LIN {X 0,Y 572.963,Z 548.941,A -85,B 0,C 180,E1 -2254.928,E2 -2254.928} C_VEL
LIN {X 0,Y 573.068,Z 542.866,A -85,B 0,C 180,E1 -2256.162,E2 -2256.162} C_VEL
LIN {X 0,Y 573.121,Z 536.225,A -85,B 0,C 180,E1 -2257.223,E2 -2257.223} C_VEL
LIN {X 0,Y 573.193,Z 527.976,A -85,B 0,C 180,E1 -2258.285,E2 -2258.285} C_VEL
LIN {X 0,Y 573.321,Z 517.583,A -85,B 0,C 180,E1 -2259.349,E2 -2259.349} C_VEL
LIN {X 0,Y 573.439,Z 507.903,A -85,B 0,C 180,E1 -2260.149,E2 -2260.149} C_VEL
LIN {X 0,Y 573.55,Z 497.379,A -85,B 0,C 180,E1 -2260.856,E2 -2260.856} C_VEL
LIN {X 0,Y 573.652,Z 485.088,A -85,B 0,C 180,E1 -2261.502,E2 -2261.502} C_VEL
LIN {X 0,Y 573.708,Z 473.128,A -85,B 0,C 180,E1 -2261.977,E2 -2261.977} C_VEL
LIN {X 0,Y 573.816,Z 460.458,A -85,B 0,C 180,E1 -2262.333,E2 -2262.333} C_VEL
LIN {X 0,Y 573.909,Z 447.193,A -85,B 0,C 180,E1 -2262.556,E2 -2262.556} C_VEL
LIN {X 0,Y 573.954,Z 350.61,A -85,B 0,C 180,E1 -2263.77,E2 -2263.77} C_VEL
LIN {X 0,Y 573.392,Z 346.603,A -85,B 0,C 180,E1 -2263.852,E2 -2263.852} C_VEL
LIN {X 0,Y 573.571,Z 326.113,A -85,B 0,C 180,E1 -2266.728,E2 -2266.728} C_VEL
LIN {X 0,Y 573.806,Z 305.604,A -85,B 0,C 180,E1 -2269.647,E2 -2269.647} C_VEL
LIN {X 0,Y 574.031,Z 285.779,A -85,B 0,C 180,E1 -2272.496,E2 -2272.496} C_VEL
LIN {X 0,Y 573.584,Z 280.847,A -85,B 0,C 180,E1 -2273.225,E2 -2273.225} C_VEL
LIN {X 0,Y 573.243,Z 279.081,A -85,B 0,C 180,E1 -2273.497,E2 -2273.497} C_VEL
LIN {X 0,Y 573.263,Z 279.079,A -85,B 0,C 180,E1 -2276.19,E2 -2276.19} C_VEL
LIN {X 0,Y 573.238,Z 279.077,A -85,B 0,C 180,E1 -2278.565,E2 -2278.565} C_VEL
LIN {X 0,Y 573.228,Z 279.075,A -85,B 0,C 180,E1 -2280.993,E2 -2280.993} C_VEL
LIN {X 0,Y 573.265,Z 279.072,A -85,B 0,C 180,E1 -2283.524,E2 -2283.524} C_VEL
LIN {X 0,Y 573.216,Z 279.084,A -85,B 0,C 180,E1 -2286.051,E2 -2286.051} C_VEL
LIN {X 0,Y 573.242,Z 279.076,A -85,B 0,C 180,E1 -2288.701,E2 -2288.701} C_VEL
LIN {X 0,Y 573.243,Z 279.073,A -85,B 0,C 180,E1 -2291.594,E2 -2291.594} C_VEL
LIN {X 0,Y 573.222,Z 279.085,A -85,B 0,C 180,E1 -2294.334,E2 -2294.334} C_VEL
LIN {X 0,Y 573.237,Z 279.074,A -85,B 0,C 180,E1 -2297.358,E2 -2297.358} C_VEL
LIN {X 0,Y 573.242,Z 279.081,A -85,B 0,C 180,E1 -2300.392,E2 -2300.392} C_VEL
LIN {X 0,Y 573.25,Z 279.075,A -85,B 0,C 180,E1 -2303.077,E2 -2303.077} C_VEL
LIN {X 0,Y 573.261,Z 279.07,A -85,B 0,C 180,E1 -2305.671,E2 -2305.671} C_VEL
LIN {X 0,Y 573.241,Z 279.075,A -85,B 0,C 180,E1 -2308.184,E2 -2308.184} C_VEL
LIN {X 0,Y 573.26,Z 279.079,A -85,B 0,C 180,E1 -2310.634,E2 -2310.634} C_VEL
LIN {X 0,Y 573.262,Z 279.072,A -85,B 0,C 180,E1 -2313.5,E2 -2313.5} C_VEL
LIN {X 0,Y 573.222,Z 279.076,A -85,B 0,C 180,E1 -2316.134,E2 -2316.134} C_VEL
LIN {X 0,Y 573.238,Z 279.081,A -85,B 0,C 180,E1 -2319.173,E2 -2319.173} C_VEL
LIN {X 0,Y 573.216,Z 279.081,A -85,B 0,C 180,E1 -2321.411,E2 -2321.411} C_VEL
LIN {X 0,Y 573.235,Z 279.076,A -85,B 0,C 180,E1 -2323.621,E2 -2323.621} C_VEL
LIN {X 0,Y 573.259,Z 279.072,A -85,B 0,C 180,E1 -2325.807,E2 -2325.807} C_VEL
LIN {X 0,Y 573.27,Z 279.072,A -85,B 0,C 180,E1 -2328.734,E2 -2328.734} C_VEL
LIN {X 0,Y 573.264,Z 279.076,A -85,B 0,C 180,E1 -2331.54,E2 -2331.54} C_VEL
LIN {X 0,Y 573.275,Z 279.069,A -85,B 0,C 180,E1 -2334.372,E2 -2334.372} C_VEL
LIN {X 0,Y 573.303,Z 279.072,A -85,B 0,C 180,E1 -2337.189,E2 -2337.189} C_VEL
LIN {X 0,Y 573.294,Z 279.069,A -85,B 0,C 180,E1 -2340,E2 -2340} C_VEL
LIN {X 0,Y 573.287,Z 279.068,A -85,B 0,C 180,E1 -2342.811,E2 -2342.811} C_VEL
LIN {X 0,Y 573.277,Z 279.08,A -85,B 0,C 180,E1 -2345.628,E2 -2345.628} C_VEL
LIN {X 0,Y 573.238,Z 279.074,A -85,B 0,C 180,E1 -2348.46,E2 -2348.46} C_VEL
LIN {X 0,Y 573.258,Z 279.074,A -85,B 0,C 180,E1 -2351.312,E2 -2351.312} C_VEL
LIN {X 0,Y 573.246,Z 279.074,A -85,B 0,C 180,E1 -2354.416,E2 -2354.416} C_VEL
LIN {X 0,Y 573.237,Z 279.074,A -85,B 0,C 180,E1 -2357.112,E2 -2357.112} C_VEL
LIN {X 0,Y 573.222,Z 279.084,A -85,B 0,C 180,E1 -2360.078,E2 -2360.078} C_VEL
LIN {X 0,Y 573.206,Z 279.082,A -85,B 0,C 180,E1 -2362.339,E2 -2362.339} C_VEL
LIN {X 0,Y 573.21,Z 279.079,A -85,B 0,C 180,E1 -2364.365,E2 -2364.365} C_VEL
LIN {X 0,Y 572.569,Z 279.16,A -85,B 0,C 180,E1 -2364.951,E2 -2364.951} C_VEL
LIN {X 0,Y 569.724,Z 279.518,A -85,B 0,C 180,E1 -2365.903,E2 -2365.903} C_VEL
LIN {X 0,Y 567.294,Z 279.816,A -85,B 0,C 180,E1 -2366.668,E2 -2366.668} C_VEL
LIN {X 0,Y 566.235,Z 279.946,A -85,B 0,C 180,E1 -2367.259,E2 -2367.259} C_VEL
LIN {X 0,Y 566.142,Z 279.958,A -85,B 0,C 180,E1 -2367.459,E2 -2367.459} C_VEL
LIN {X 0,Y 566.163,Z 279.959,A -85,B 0,C 180,E1 -2370.594,E2 -2370.594} C_VEL
LIN {X 0,Y 566.19,Z 279.952,A -85,B 0,C 180,E1 -2373.104,E2 -2373.104} C_VEL
LIN {X 0,Y 566.129,Z 279.96,A -85,B 0,C 180,E1 -2375.695,E2 -2375.695} C_VEL
LIN {X 0,Y 566.191,Z 279.959,A -85,B 0,C 180,E1 -2378.557,E2 -2378.557} C_VEL
LIN {X 0,Y 566.124,Z 279.961,A -85,B 0,C 180,E1 -2381.144,E2 -2381.144} C_VEL
LIN {X 0,Y 566.141,Z 279.96,A -85,B 0,C 180,E1 -2384.042,E2 -2384.042} C_VEL
LIN {X 0,Y 566.138,Z 279.961,A -85,B 0,C 180,E1 -2387.09,E2 -2387.09} C_VEL
LIN {X 0,Y 566.171,Z 279.958,A -85,B 0,C 180,E1 -2390.32,E2 -2390.32} C_VEL
LIN {X 0,Y 566.136,Z 279.959,A -85,B 0,C 180,E1 -2393.425,E2 -2393.425} C_VEL
LIN {X 0,Y 566.144,Z 279.959,A -85,B 0,C 180,E1 -2396.277,E2 -2396.277} C_VEL
LIN {X 0,Y 566.166,Z 279.965,A -85,B 0,C 180,E1 -2398.928,E2 -2398.928} C_VEL
LIN {X 0,Y 566.143,Z 279.957,A -85,B 0,C 180,E1 -2401.853,E2 -2401.853} C_VEL
LIN {X 0,Y 566.164,Z 279.955,A -85,B 0,C 180,E1 -2404.248,E2 -2404.248} C_VEL
LIN {X 0,Y 566.154,Z 279.962,A -85,B 0,C 180,E1 -2407.367,E2 -2407.367} C_VEL
LIN {X 0,Y 566.202,Z 279.952,A -85,B 0,C 180,E1 -2409.661,E2 -2409.661} C_VEL
LIN {X 0,Y 566.176,Z 279.955,A -85,B 0,C 180,E1 -2412.666,E2 -2412.666} C_VEL
LIN {X 0,Y 566.214,Z 279.953,A -85,B 0,C 180,E1 -2415.625,E2 -2415.625} C_VEL
LIN {X 0,Y 566.24,Z 279.946,A -85,B 0,C 180,E1 -2418.675,E2 -2418.675} C_VEL
LIN {X 0,Y 566.193,Z 279.962,A -85,B 0,C 180,E1 -2421.432,E2 -2421.432} C_VEL
LIN {X 0,Y 566.234,Z 279.946,A -85,B 0,C 180,E1 -2424.3,E2 -2424.3} C_VEL
LIN {X 0,Y 566.278,Z 279.946,A -85,B 0,C 180,E1 -2427.864,E2 -2427.864} C_VEL
LIN {X 0,Y 566.288,Z 279.944,A -85,B 0,C 180,E1 -2429.998,E2 -2429.998} C_VEL
LIN {X 0,Y 566.247,Z 279.944,A -85,B 0,C 180,E1 -2432.843,E2 -2432.843} C_VEL
LIN {X 0,Y 566.244,Z 279.954,A -85,B 0,C 180,E1 -2435.696,E2 -2435.696} C_VEL
LIN {X 0,Y 566.201,Z 279.952,A -85,B 0,C 180,E1 -2438.563,E2 -2438.563} C_VEL
LIN {X 0,Y 566.194,Z 279.956,A -85,B 0,C 180,E1 -2441.452,E2 -2441.452} C_VEL
LIN {X 0,Y 566.245,Z 280.006,A -85,B 0,C 180,E1 -2442.86,E2 -2442.86} C_VEL
LIN {X 0,Y 566.448,Z 288.153,A -85,B 0,C 180,E1 -2444.364,E2 -2444.364} C_VEL
LIN {X 0,Y 566.29,Z 303.331,A -85,B 0,C 180,E1 -2447.133,E2 -2447.133} C_VEL
LIN {X 0,Y 566.23,Z 308.399,A -85,B 0,C 180,E1 -2448.05,E2 -2448.05} C_VEL
LIN {X 0,Y 567.175,Z 314.711,A -85,B 0,C 180,E1 -2448.159,E2 -2448.159} C_VEL
LIN {X 0,Y 566.915,Z 415.457,A -85,B 0,C 180,E1 -2449.457,E2 -2449.457} C_VEL
LIN {X 0,Y 566.84,Z 428.654,A -85,B 0,C 180,E1 -2449.777,E2 -2449.777} C_VEL
LIN {X 0,Y 566.74,Z 440.771,A -85,B 0,C 180,E1 -2450.209,E2 -2450.209} C_VEL
LIN {X 0,Y 566.578,Z 452.89,A -85,B 0,C 180,E1 -2450.794,E2 -2450.794} C_VEL
LIN {X 0,Y 566.394,Z 463.739,A -85,B 0,C 180,E1 -2451.467,E2 -2451.467} C_VEL
LIN {X 0,Y 566.282,Z 474.893,A -85,B 0,C 180,E1 -2452.334,E2 -2452.334} C_VEL
LIN {X 0,Y 566.196,Z 484.666,A -85,B 0,C 180,E1 -2453.286,E2 -2453.286} C_VEL
LIN {X 0,Y 566.085,Z 493.699,A -85,B 0,C 180,E1 -2454.377,E2 -2454.377} C_VEL
LIN {X 0,Y 565.999,Z 500.298,A -85,B 0,C 180,E1 -2455.36,E2 -2455.36} C_VEL
LIN {X 0,Y 565.956,Z 506.681,A -85,B 0,C 180,E1 -2456.55,E2 -2456.55} C_VEL
LIN {X 0,Y 565.879,Z 511.585,A -85,B 0,C 180,E1 -2457.745,E2 -2457.745} C_VEL
LIN {X 0,Y 565.883,Z 515.239,A -85,B 0,C 180,E1 -2458.966,E2 -2458.966} C_VEL
LIN {X 0,Y 565.858,Z 516.997,A -85,B 0,C 180,E1 -2459.784,E2 -2459.784} C_VEL
LIN {X 0,Y 565.856,Z 518.576,A -85,B 0,C 180,E1 -2461.019,E2 -2461.019} C_VEL
LIN {X 0,Y 565.833,Z 518.934,A -85,B 0,C 180,E1 -2462.37,E2 -2462.37} C_VEL
LIN {X 0,Y 565.863,Z 517.946,A -85,B 0,C 180,E1 -2463.681,E2 -2463.681} C_VEL
LIN {X 0,Y 565.848,Z 515.692,A -85,B 0,C 180,E1 -2464.941,E2 -2464.941} C_VEL
LIN {X 0,Y 565.913,Z 512.179,A -85,B 0,C 180,E1 -2466.174,E2 -2466.174} C_VEL
LIN {X 0,Y 565.949,Z 506.981,A -85,B 0,C 180,E1 -2467.474,E2 -2467.474} C_VEL
LIN {X 0,Y 565.992,Z 500.618,A -85,B 0,C 180,E1 -2468.678,E2 -2468.678} C_VEL
LIN {X 0,Y 566.057,Z 494.058,A -85,B 0,C 180,E1 -2469.666,E2 -2469.666} C_VEL
LIN {X 0,Y 566.174,Z 484.874,A -85,B 0,C 180,E1 -2470.782,E2 -2470.782} C_VEL
LIN {X 0,Y 566.318,Z 475.145,A -85,B 0,C 180,E1 -2471.734,E2 -2471.734} C_VEL
LIN {X 0,Y 566.41,Z 464.873,A -85,B 0,C 180,E1 -2472.543,E2 -2472.543} C_VEL
LIN {X 0,Y 566.558,Z 453.576,A -85,B 0,C 180,E1 -2473.257,E2 -2473.257} C_VEL
LIN {X 0,Y 566.73,Z 441.453,A -85,B 0,C 180,E1 -2473.853,E2 -2473.853} C_VEL
LIN {X 0,Y 566.855,Z 428.486,A -85,B 0,C 180,E1 -2474.318,E2 -2474.318} C_VEL
LIN {X 0,Y 566.929,Z 414.948,A -85,B 0,C 180,E1 -2474.643,E2 -2474.643} C_VEL
LIN {X 0,Y 567.03,Z 313.172,A -85,B 0,C 180,E1 -2475.954,E2 -2475.954} C_VEL
LIN {X 0,Y 566.221,Z 308.405,A -85,B 0,C 180,E1 -2476.039,E2 -2476.039} C_VEL
LIN {X 0,Y 566.38,Z 293.821,A -85,B 0,C 180,E1 -2478.687,E2 -2478.687} C_VEL
LIN {X 0,Y 566.4,Z 281.479,A -85,B 0,C 180,E1 -2480.935,E2 -2480.935} C_VEL
LIN {X 0,Y 566.214,Z 279.954,A -85,B 0,C 180,E1 -2481.208,E2 -2481.208} C_VEL
LIN {X 0,Y 566.173,Z 279.964,A -85,B 0,C 180,E1 -2484.308,E2 -2484.308} C_VEL
LIN {X 0,Y 566.186,Z 279.954,A -85,B 0,C 180,E1 -2486.895,E2 -2486.895} C_VEL
LIN {X 0,Y 566.151,Z 279.957,A -85,B 0,C 180,E1 -2489.405,E2 -2489.405} C_VEL
LIN {X 0,Y 566.18,Z 279.956,A -85,B 0,C 180,E1 -2491.856,E2 -2491.856} C_VEL
LIN {X 0,Y 566.185,Z 279.962,A -85,B 0,C 180,E1 -2494.249,E2 -2494.249} C_VEL
LIN {X 0,Y 566.143,Z 279.965,A -85,B 0,C 180,E1 -2496.71,E2 -2496.71} C_VEL
LIN {X 0,Y 566.162,Z 279.956,A -85,B 0,C 180,E1 -2499.661,E2 -2499.661} C_VEL
LIN {X 0,Y 566.15,Z 279.965,A -85,B 0,C 180,E1 -2502.667,E2 -2502.667} C_VEL
LIN {X 0,Y 566.178,Z 279.953,A -85,B 0,C 180,E1 -2505.625,E2 -2505.625} C_VEL
LIN {X 0,Y 566.22,Z 279.958,A -85,B 0,C 180,E1 -2508.652,E2 -2508.652} C_VEL
LIN {X 0,Y 566.176,Z 279.954,A -85,B 0,C 180,E1 -2511.433,E2 -2511.433} C_VEL
LIN {X 0,Y 566.214,Z 279.952,A -85,B 0,C 180,E1 -2514.301,E2 -2514.301} C_VEL
LIN {X 0,Y 566.226,Z 279.952,A -85,B 0,C 180,E1 -2517.154,E2 -2517.154} C_VEL
LIN {X 0,Y 566.225,Z 279.946,A -85,B 0,C 180,E1 -2520,E2 -2520} C_VEL
LIN {X 0,Y 566.233,Z 279.956,A -85,B 0,C 180,E1 -2522.846,E2 -2522.846} C_VEL
LIN {X 0,Y 566.218,Z 279.949,A -85,B 0,C 180,E1 -2525.699,E2 -2525.699} C_VEL
LIN {X 0,Y 566.2,Z 279.952,A -85,B 0,C 180,E1 -2528.566,E2 -2528.566} C_VEL
LIN {X 0,Y 566.209,Z 279.952,A -85,B 0,C 180,E1 -2531.455,E2 -2531.455} C_VEL
LIN {X 0,Y 566.179,Z 279.954,A -85,B 0,C 180,E1 -2534.509,E2 -2534.509} C_VEL
LIN {X 0,Y 566.17,Z 279.962,A -85,B 0,C 180,E1 -2537.333,E2 -2537.333} C_VEL
LIN {X 0,Y 566.176,Z 279.952,A -85,B 0,C 180,E1 -2540.339,E2 -2540.339} C_VEL
LIN {X 0,Y 566.199,Z 279.958,A -85,B 0,C 180,E1 -2543.404,E2 -2543.404} C_VEL
LIN {X 0,Y 566.188,Z 279.956,A -85,B 0,C 180,E1 -2545.75,E2 -2545.75} C_VEL
LIN {X 0,Y 566.2,Z 279.95,A -85,B 0,C 180,E1 -2548.214,E2 -2548.214} C_VEL
LIN {X 0,Y 566.165,Z 279.959,A -85,B 0,C 180,E1 -2551.083,E2 -2551.083} C_VEL
LIN {X 0,Y 566.185,Z 279.955,A -85,B 0,C 180,E1 -2553.958,E2 -2553.958} C_VEL
LIN {X 0,Y 566.183,Z 279.953,A -85,B 0,C 180,E1 -2556.571,E2 -2556.571} C_VEL
LIN {X 0,Y 566.237,Z 279.955,A -85,B 0,C 180,E1 -2559.697,E2 -2559.697} C_VEL
LIN {X 0,Y 566.196,Z 279.955,A -85,B 0,C 180,E1 -2562.089,E2 -2562.089} C_VEL
LIN {X 0,Y 566.141,Z 279.96,A -85,B 0,C 180,E1 -2565.039,E2 -2565.039} C_VEL
LIN {X 0,Y 566.202,Z 279.955,A -85,B 0,C 180,E1 -2568.138,E2 -2568.138} C_VEL
LIN {X 0,Y 566.201,Z 279.951,A -85,B 0,C 180,E1 -2570.732,E2 -2570.732} C_VEL
LIN {X 0,Y 566.196,Z 279.961,A -85,B 0,C 180,E1 -2573.787,E2 -2573.787} C_VEL
LIN {X 0,Y 566.209,Z 279.955,A -85,B 0,C 180,E1 -2576.267,E2 -2576.267} C_VEL
LIN {X 0,Y 566.187,Z 279.954,A -85,B 0,C 180,E1 -2578.925,E2 -2578.925} C_VEL
LIN {X 0,Y 566.182,Z 279.954,A -85,B 0,C 180,E1 -2581.051,E2 -2581.051} C_VEL
LIN {X 0,Y 566.234,Z 279.95,A -85,B 0,C 180,E1 -2583.464,E2 -2583.464} C_VEL
LIN {X 0,Y 566.227,Z 279.974,A -85,B 0,C 180,E1 -2586.408,E2 -2586.408} C_VEL
LIN {X 0,Y 567.052,Z 285.349,A -85,B 0,C 180,E1 -2587.217,E2 -2587.217} C_VEL
LIN {X 0,Y 566.864,Z 306.734,A -85,B 0,C 180,E1 -2590.277,E2 -2590.277} C_VEL
LIN {X 0,Y 566.593,Z 327.574,A -85,B 0,C 180,E1 -2593.269,E2 -2593.269} C_VEL
LIN {X 0,Y 566.402,Z 346.718,A -85,B 0,C 180,E1 -2595.99,E2 -2595.99} C_VEL
LIN {X 0,Y 567.163,Z 353.503,A -85,B 0,C 180,E1 -2596.098,E2 -2596.098} C_VEL
LIN {X 0,Y 566.948,Z 455.109,A -85,B 0,C 180,E1 -2597.406,E2 -2597.406} C_VEL
LIN {X 0,Y 566.813,Z 468.326,A -85,B 0,C 180,E1 -2597.721,E2 -2597.721} C_VEL
LIN {X 0,Y 566.726,Z 480.456,A -85,B 0,C 180,E1 -2598.151,E2 -2598.151} C_VEL
LIN {X 0,Y 566.623,Z 492.12,A -85,B 0,C 180,E1 -2598.706,E2 -2598.706} C_VEL
LIN {X 0,Y 566.486,Z 502.951,A -85,B 0,C 180,E1 -2599.369,E2 -2599.369} C_VEL
LIN {X 0,Y 566.328,Z 513.575,A -85,B 0,C 180,E1 -2600.178,E2 -2600.178} C_VEL
LIN {X 0,Y 566.204,Z 523.111,A -85,B 0,C 180,E1 -2601.077,E2 -2601.077} C_VEL
LIN {X 0,Y 566.11,Z 530.984,A -85,B 0,C 180,E1 -2601.975,E2 -2601.975} C_VEL
LIN {X 0,Y 566.02,Z 538.64,A -85,B 0,C 180,E1 -2603.05,E2 -2603.05} C_VEL
LIN {X 0,Y 566.005,Z 545.694,A -85,B 0,C 180,E1 -2604.302,E2 -2604.302} C_VEL
LIN {X 0,Y 565.933,Z 550.383,A -85,B 0,C 180,E1 -2605.373,E2 -2605.373} C_VEL
LIN {X 0,Y 565.926,Z 553.965,A -85,B 0,C 180,E1 -2606.443,E2 -2606.443} C_VEL
LIN {X 0,Y 565.877,Z 555.814,A -85,B 0,C 180,E1 -2607.155,E2 -2607.155} C_VEL
LIN {X 0,Y 565.845,Z 558.188,A -85,B 0,C 180,E1 -2608.579,E2 -2608.579} C_VEL
LIN {X 0,Y 565.839,Z 559,A -85,B 0,C 180,E1 -2610.002,E2 -2610.002} C_VEL
LIN {X 0,Y 565.845,Z 558.183,A -85,B 0,C 180,E1 -2611.426,E2 -2611.426} C_VEL
LIN {X 0,Y 565.878,Z 555.805,A -85,B 0,C 180,E1 -2612.85,E2 -2612.85} C_VEL
LIN {X 0,Y 565.926,Z 552.889,A -85,B 0,C 180,E1 -2613.919,E2 -2613.919} C_VEL
LIN {X 0,Y 565.878,Z 548.941,A -85,B 0,C 180,E1 -2614.989,E2 -2614.989} C_VEL
LIN {X 0,Y 565.995,Z 542.866,A -85,B 0,C 180,E1 -2616.239,E2 -2616.239} C_VEL
LIN {X 0,Y 566.054,Z 536.224,A -85,B 0,C 180,E1 -2617.313,E2 -2617.313} C_VEL
LIN {X 0,Y 566.142,Z 527.977,A -85,B 0,C 180,E1 -2618.389,E2 -2618.389} C_VEL
LIN {X 0,Y 566.255,Z 519.521,A -85,B 0,C 180,E1 -2619.287,E2 -2619.287} C_VEL
LIN {X 0,Y 566.394,Z 509.075,A -85,B 0,C 180,E1 -2620.186,E2 -2620.186} C_VEL
LIN {X 0,Y 566.571,Z 497.68,A -85,B 0,C 180,E1 -2620.972,E2 -2620.972} C_VEL
LIN {X 0,Y 566.694,Z 485.852,A -85,B 0,C 180,E1 -2621.61,E2 -2621.61} C_VEL
LIN {X 0,Y 566.778,Z 473.126,A -85,B 0,C 180,E1 -2622.125,E2 -2622.125} C_VEL
LIN {X 0,Y 566.903,Z 460.457,A -85,B 0,C 180,E1 -2622.486,E2 -2622.486} C_VEL
LIN {X 0,Y 566.977,Z 447.193,A -85,B 0,C 180,E1 -2622.712,E2 -2622.712} C_VEL
LIN {X 0,Y 567.049,Z 351.169,A -85,B 0,C 180,E1 -2623.934,E2 -2623.934} C_VEL
LIN {X 0,Y 566.386,Z 346.603,A -85,B 0,C 180,E1 -2624.027,E2 -2624.027} C_VEL
LIN {X 0,Y 566.614,Z 324.883,A -85,B 0,C 180,E1 -2627.116,E2 -2627.116} C_VEL
LIN {X 0,Y 566.87,Z 303.961,A -85,B 0,C 180,E1 -2630.124,E2 -2630.124} C_VEL
LIN {X 0,Y 567.061,Z 285.545,A -85,B 0,C 180,E1 -2632.788,E2 -2632.788} C_VEL
LIN {X 0,Y 566.209,Z 279.958,A -85,B 0,C 180,E1 -2633.646,E2 -2633.646} C_VEL
LIN {X 0,Y 566.212,Z 279.958,A -85,B 0,C 180,E1 -2635.75,E2 -2635.75} C_VEL
LIN {X 0,Y 566.207,Z 279.958,A -85,B 0,C 180,E1 -2638.202,E2 -2638.202} C_VEL
LIN {X 0,Y 566.193,Z 279.952,A -85,B 0,C 180,E1 -2641.076,E2 -2641.076} C_VEL
LIN {X 0,Y 566.214,Z 279.952,A -85,B 0,C 180,E1 -2643.734,E2 -2643.734} C_VEL
LIN {X 0,Y 566.201,Z 279.955,A -85,B 0,C 180,E1 -2646.57,E2 -2646.57} C_VEL
LIN {X 0,Y 566.215,Z 279.95,A -85,B 0,C 180,E1 -2649.685,E2 -2649.685} C_VEL
LIN {X 0,Y 566.21,Z 279.955,A -85,B 0,C 180,E1 -2652.087,E2 -2652.087} C_VEL
LIN {X 0,Y 566.165,Z 279.956,A -85,B 0,C 180,E1 -2655.036,E2 -2655.036} C_VEL
LIN {X 0,Y 566.215,Z 279.953,A -85,B 0,C 180,E1 -2658.135,E2 -2658.135} C_VEL
LIN {X 0,Y 566.216,Z 279.956,A -85,B 0,C 180,E1 -2660.726,E2 -2660.726} C_VEL
LIN {X 0,Y 566.2,Z 279.95,A -85,B 0,C 180,E1 -2663.785,E2 -2663.785} C_VEL
LIN {X 0,Y 566.222,Z 279.955,A -85,B 0,C 180,E1 -2666.898,E2 -2666.898} C_VEL
LIN {X 0,Y 566.185,Z 279.953,A -85,B 0,C 180,E1 -2669.407,E2 -2669.407} C_VEL
LIN {X 0,Y 566.203,Z 279.95,A -85,B 0,C 180,E1 -2671.857,E2 -2671.857} C_VEL
LIN {X 0,Y 566.216,Z 279.95,A -85,B 0,C 180,E1 -2674.251,E2 -2674.251} C_VEL
LIN {X 0,Y 566.181,Z 279.959,A -85,B 0,C 180,E1 -2676.713,E2 -2676.713} C_VEL
LIN {X 0,Y 566.201,Z 279.951,A -85,B 0,C 180,E1 -2679.662,E2 -2679.662} C_VEL
LIN {X 0,Y 566.187,Z 279.956,A -85,B 0,C 180,E1 -2682.668,E2 -2682.668} C_VEL
LIN {X 0,Y 566.22,Z 279.951,A -85,B 0,C 180,E1 -2685.626,E2 -2685.626} C_VEL
LIN {X 0,Y 566.229,Z 279.949,A -85,B 0,C 180,E1 -2688.671,E2 -2688.671} C_VEL
LIN {X 0,Y 566.211,Z 279.957,A -85,B 0,C 180,E1 -2691.434,E2 -2691.434} C_VEL
LIN {X 0,Y 566.242,Z 279.945,A -85,B 0,C 180,E1 -2694.302,E2 -2694.302} C_VEL
LIN {X 0,Y 566.268,Z 279.948,A -85,B 0,C 180,E1 -2697.154,E2 -2697.154} C_VEL
LIN {X 0,Y 566.265,Z 279.945,A -85,B 0,C 180,E1 -2700,E2 -2700} C_VEL
LIN {X 0,Y 566.254,Z 279.944,A -85,B 0,C 180,E1 -2702.846,E2 -2702.846} C_VEL
LIN {X 0,Y 566.242,Z 279.954,A -85,B 0,C 180,E1 -2705.699,E2 -2705.699} C_VEL
LIN {X 0,Y 566.189,Z 279.952,A -85,B 0,C 180,E1 -2708.566,E2 -2708.566} C_VEL
LIN {X 0,Y 566.228,Z 279.952,A -85,B 0,C 180,E1 -2711.455,E2 -2711.455} C_VEL
LIN {X 0,Y 566.202,Z 279.951,A -85,B 0,C 180,E1 -2714.499,E2 -2714.499} C_VEL
LIN {X 0,Y 566.181,Z 279.955,A -85,B 0,C 180,E1 -2717.332,E2 -2717.332} C_VEL
LIN {X 0,Y 566.189,Z 279.956,A -85,B 0,C 180,E1 -2720.338,E2 -2720.338} C_VEL
LIN {X 0,Y 566.154,Z 279.956,A -85,B 0,C 180,E1 -2723.28,E2 -2723.28} C_VEL
LIN {X 0,Y 566.18,Z 279.957,A -85,B 0,C 180,E1 -2725.751,E2 -2725.751} C_VEL
LIN {X 0,Y 566.142,Z 279.958,A -85,B 0,C 180,E1 -2727.459,E2 -2727.459} C_VEL
LIN {X 0,Y 565.458,Z 280.052,A -85,B 0,C 180,E1 -2728.053,E2 -2728.053} C_VEL
LIN {X 0,Y 562.605,Z 280.409,A -85,B 0,C 180,E1 -2729.017,E2 -2729.017} C_VEL
LIN {X 0,Y 560.213,Z 280.706,A -85,B 0,C 180,E1 -2729.793,E2 -2729.793} C_VEL
LIN {X 0,Y 559.197,Z 280.83,A -85,B 0,C 180,E1 -2730.392,E2 -2730.392} C_VEL
LIN {X 0,Y 559.119,Z 280.836,A -85,B 0,C 180,E1 -2730.594,E2 -2730.594} C_VEL
LIN {X 0,Y 559.142,Z 280.833,A -85,B 0,C 180,E1 -2732.716,E2 -2732.716} C_VEL
LIN {X 0,Y 559.106,Z 280.834,A -85,B 0,C 180,E1 -2735.326,E2 -2735.326} C_VEL
LIN {X 0,Y 559.115,Z 280.837,A -85,B 0,C 180,E1 -2738.019,E2 -2738.019} C_VEL
LIN {X 0,Y 559.082,Z 280.841,A -85,B 0,C 180,E1 -2740.819,E2 -2740.819} C_VEL
LIN {X 0,Y 559.088,Z 280.837,A -85,B 0,C 180,E1 -2743.191,E2 -2743.191} C_VEL
LIN {X 0,Y 559.109,Z 280.834,A -85,B 0,C 180,E1 -2745.766,E2 -2745.766} C_VEL
LIN {X 0,Y 559.089,Z 280.84,A -85,B 0,C 180,E1 -2748.223,E2 -2748.223} C_VEL
LIN {X 0,Y 559.103,Z 280.839,A -85,B 0,C 180,E1 -2751.06,E2 -2751.06} C_VEL
LIN {X 0,Y 559.105,Z 280.834,A -85,B 0,C 180,E1 -2753.787,E2 -2753.787} C_VEL
LIN {X 0,Y 559.092,Z 280.839,A -85,B 0,C 180,E1 -2756.42,E2 -2756.42} C_VEL
LIN {X 0,Y 559.132,Z 280.84,A -85,B 0,C 180,E1 -2758.979,E2 -2758.979} C_VEL
LIN {X 0,Y 559.101,Z 280.835,A -85,B 0,C 180,E1 -2762.283,E2 -2762.283} C_VEL
LIN {X 0,Y 559.118,Z 280.839,A -85,B 0,C 180,E1 -2764.827,E2 -2764.827} C_VEL
LIN {X 0,Y 559.129,Z 280.832,A -85,B 0,C 180,E1 -2767.846,E2 -2767.846} C_VEL
LIN {X 0,Y 559.165,Z 280.828,A -85,B 0,C 180,E1 -2770.503,E2 -2770.503} C_VEL
LIN {X 0,Y 559.147,Z 280.839,A -85,B 0,C 180,E1 -2773.195,E2 -2773.195} C_VEL
LIN {X 0,Y 559.149,Z 280.829,A -85,B 0,C 180,E1 -2776.182,E2 -2776.182} C_VEL
LIN {X 0,Y 559.185,Z 280.83,A -85,B 0,C 180,E1 -2779.132,E2 -2779.132} C_VEL
LIN {X 0,Y 559.141,Z 280.831,A -85,B 0,C 180,E1 -2782.051,E2 -2782.051} C_VEL
LIN {X 0,Y 559.239,Z 280.819,A -85,B 0,C 180,E1 -2784.951,E2 -2784.951} C_VEL
LIN {X 0,Y 559.249,Z 280.822,A -85,B 0,C 180,E1 -2787.837,E2 -2787.837} C_VEL
LIN {X 0,Y 559.257,Z 280.819,A -85,B 0,C 180,E1 -2789.998,E2 -2789.998} C_VEL
LIN {X 0,Y 559.215,Z 280.821,A -85,B 0,C 180,E1 -2792.879,E2 -2792.879} C_VEL
LIN {X 0,Y 559.213,Z 280.832,A -85,B 0,C 180,E1 -2795.768,E2 -2795.768} C_VEL
LIN {X 0,Y 559.164,Z 280.828,A -85,B 0,C 180,E1 -2798.672,E2 -2798.672} C_VEL
LIN {X 0,Y 559.162,Z 280.835,A -85,B 0,C 180,E1 -2801.598,E2 -2801.598} C_VEL
LIN {X 0,Y 559.204,Z 280.884,A -85,B 0,C 180,E1 -2802.794,E2 -2802.794} C_VEL
LIN {X 0,Y 559.45,Z 288.313,A -85,B 0,C 180,E1 -2804.176,E2 -2804.176} C_VEL
LIN {X 0,Y 559.278,Z 303.723,A -85,B 0,C 180,E1 -2807.014,E2 -2807.014} C_VEL
LIN {X 0,Y 559.21,Z 308.42,A -85,B 0,C 180,E1 -2807.875,E2 -2807.875} C_VEL
LIN {X 0,Y 560.302,Z 315.754,A -85,B 0,C 180,E1 -2807.999,E2 -2807.999} C_VEL
LIN {X 0,Y 560.001,Z 415.075,A -85,B 0,C 180,E1 -2809.292,E2 -2809.292} C_VEL
LIN {X 0,Y 559.902,Z 428.924,A -85,B 0,C 180,E1 -2809.631,E2 -2809.631} C_VEL
LIN {X 0,Y 559.771,Z 441.696,A -85,B 0,C 180,E1 -2810.098,E2 -2810.098} C_VEL
LIN {X 0,Y 559.595,Z 453.389,A -85,B 0,C 180,E1 -2810.681,E2 -2810.681} C_VEL
LIN {X 0,Y 559.394,Z 465.23,A -85,B 0,C 180,E1 -2811.439,E2 -2811.439} C_VEL
LIN {X 0,Y 559.261,Z 475.235,A -85,B 0,C 180,E1 -2812.241,E2 -2812.241} C_VEL
LIN {X 0,Y 559.145,Z 485.095,A -85,B 0,C 180,E1 -2813.222,E2 -2813.222} C_VEL
LIN {X 0,Y 559.037,Z 493.916,A -85,B 0,C 180,E1 -2814.309,E2 -2814.309} C_VEL
LIN {X 0,Y 558.92,Z 501.638,A -85,B 0,C 180,E1 -2815.505,E2 -2815.505} C_VEL
LIN {X 0,Y 558.874,Z 507.959,A -85,B 0,C 180,E1 -2816.766,E2 -2816.766} C_VEL
LIN {X 0,Y 558.784,Z 511.717,A -85,B 0,C 180,E1 -2817.729,E2 -2817.729} C_VEL
LIN {X 0,Y 558.795,Z 514.27,A -85,B 0,C 180,E1 -2818.545,E2 -2818.545} C_VEL
LIN {X 0,Y 558.758,Z 517.049,A -85,B 0,C 180,E1 -2819.787,E2 -2819.787} C_VEL
LIN {X 0,Y 558.751,Z 518.708,A -85,B 0,C 180,E1 -2821.206,E2 -2821.206} C_VEL
LIN {X 0,Y 558.747,Z 518.891,A -85,B 0,C 180,E1 -2822.569,E2 -2822.569} C_VEL
LIN {X 0,Y 558.763,Z 517.692,A -85,B 0,C 180,E1 -2823.887,E2 -2823.887} C_VEL
LIN {X 0,Y 558.766,Z 515.246,A -85,B 0,C 180,E1 -2825.159,E2 -2825.159} C_VEL
LIN {X 0,Y 558.817,Z 511.586,A -85,B 0,C 180,E1 -2826.399,E2 -2826.399} C_VEL
LIN {X 0,Y 558.873,Z 506.71,A -85,B 0,C 180,E1 -2827.604,E2 -2827.604} C_VEL
LIN {X 0,Y 558.908,Z 500.549,A -85,B 0,C 180,E1 -2828.774,E2 -2828.774} C_VEL
LIN {X 0,Y 559.027,Z 492.848,A -85,B 0,C 180,E1 -2829.925,E2 -2829.925} C_VEL
LIN {X 0,Y 559.145,Z 484.551,A -85,B 0,C 180,E1 -2830.928,E2 -2830.928} C_VEL
LIN {X 0,Y 559.298,Z 475.203,A -85,B 0,C 180,E1 -2831.851,E2 -2831.851} C_VEL
LIN {X 0,Y 559.427,Z 464.369,A -85,B 0,C 180,E1 -2832.711,E2 -2832.711} C_VEL
LIN {X 0,Y 559.616,Z 452.378,A -85,B 0,C 180,E1 -2833.467,E2 -2833.467} C_VEL
LIN {X 0,Y 559.77,Z 440.879,A -85,B 0,C 180,E1 -2834.026,E2 -2834.026} C_VEL
LIN {X 0,Y 559.91,Z 427.752,A -85,B 0,C 180,E1 -2834.495,E2 -2834.495} C_VEL
LIN {X 0,Y 560.009,Z 414.89,A -85,B 0,C 180,E1 -2834.802,E2 -2834.802} C_VEL
LIN {X 0,Y 560.169,Z 314.157,A -85,B 0,C 180,E1 -2836.115,E2 -2836.115} C_VEL
LIN {X 0,Y 559.193,Z 308.368,A -85,B 0,C 180,E1 -2836.225,E2 -2836.225} C_VEL
LIN {X 0,Y 559.33,Z 293.582,A -85,B 0,C 180,E1 -2838.921,E2 -2838.921} C_VEL
LIN {X 0,Y 559.235,Z 281.283,A -85,B 0,C 180,E1 -2841.071,E2 -2841.071} C_VEL
LIN {X 0,Y 559.168,Z 280.832,A -85,B 0,C 180,E1 -2841.184,E2 -2841.184} C_VEL
LIN {X 0,Y 559.133,Z 280.836,A -85,B 0,C 180,E1 -2843.789,E2 -2843.789} C_VEL
LIN {X 0,Y 559.136,Z 280.839,A -85,B 0,C 180,E1 -2846.423,E2 -2846.423} C_VEL
LIN {X 0,Y 559.124,Z 280.834,A -85,B 0,C 180,E1 -2848.979,E2 -2848.979} C_VEL
LIN {X 0,Y 559.124,Z 280.834,A -85,B 0,C 180,E1 -2851.615,E2 -2851.615} C_VEL
LIN {X 0,Y 559.157,Z 280.832,A -85,B 0,C 180,E1 -2853.902,E2 -2853.902} C_VEL
LIN {X 0,Y 559.108,Z 280.844,A -85,B 0,C 180,E1 -2856.564,E2 -2856.564} C_VEL
LIN {X 0,Y 559.127,Z 280.833,A -85,B 0,C 180,E1 -2859.393,E2 -2859.393} C_VEL
LIN {X 0,Y 559.102,Z 280.835,A -85,B 0,C 180,E1 -2861.684,E2 -2861.684} C_VEL
LIN {X 0,Y 559.115,Z 280.835,A -85,B 0,C 180,E1 -2863.946,E2 -2863.946} C_VEL
LIN {X 0,Y 559.12,Z 280.836,A -85,B 0,C 180,E1 -2866.183,E2 -2866.183} C_VEL
LIN {X 0,Y 559.159,Z 280.83,A -85,B 0,C 180,E1 -2869.133,E2 -2869.133} C_VEL
LIN {X 0,Y 559.153,Z 280.83,A -85,B 0,C 180,E1 -2872.053,E2 -2872.053} C_VEL
LIN {X 0,Y 559.205,Z 280.828,A -85,B 0,C 180,E1 -2874.953,E2 -2874.953} C_VEL
LIN {X 0,Y 559.188,Z 280.824,A -85,B 0,C 180,E1 -2877.839,E2 -2877.839} C_VEL
LIN {X 0,Y 559.231,Z 280.825,A -85,B 0,C 180,E1 -2880.72,E2 -2880.72} C_VEL
LIN {X 0,Y 559.198,Z 280.832,A -85,B 0,C 180,E1 -2882.882,E2 -2882.882} C_VEL
LIN {X 0,Y 559.185,Z 280.825,A -85,B 0,C 180,E1 -2885.771,E2 -2885.771} C_VEL
LIN {X 0,Y 559.156,Z 280.831,A -85,B 0,C 180,E1 -2888.675,E2 -2888.675} C_VEL
LIN {X 0,Y 559.16,Z 280.828,A -85,B 0,C 180,E1 -2891.601,E2 -2891.601} C_VEL
LIN {X 0,Y 559.143,Z 280.832,A -85,B 0,C 180,E1 -2894.597,E2 -2894.597} C_VEL
LIN {X 0,Y 559.144,Z 280.834,A -85,B 0,C 180,E1 -2897.557,E2 -2897.557} C_VEL
LIN {X 0,Y 559.141,Z 280.829,A -85,B 0,C 180,E1 -2900.606,E2 -2900.606} C_VEL
LIN {X 0,Y 559.153,Z 280.835,A -85,B 0,C 180,E1 -2903.446,E2 -2903.446} C_VEL
LIN {X 0,Y 559.161,Z 280.828,A -85,B 0,C 180,E1 -2906.098,E2 -2906.098} C_VEL
LIN {X 0,Y 559.139,Z 280.829,A -85,B 0,C 180,E1 -2908.531,E2 -2908.531} C_VEL
LIN {X 0,Y 559.118,Z 280.84,A -85,B 0,C 180,E1 -2911.279,E2 -2911.279} C_VEL
LIN {X 0,Y 559.14,Z 280.833,A -85,B 0,C 180,E1 -2913.955,E2 -2913.955} C_VEL
LIN {X 0,Y 559.158,Z 280.828,A -85,B 0,C 180,E1 -2916.456,E2 -2916.456} C_VEL
LIN {X 0,Y 559.197,Z 280.829,A -85,B 0,C 180,E1 -2919.864,E2 -2919.864} C_VEL
LIN {X 0,Y 559.14,Z 280.831,A -85,B 0,C 180,E1 -2922.746,E2 -2922.746} C_VEL
LIN {X 0,Y 559.124,Z 280.843,A -85,B 0,C 180,E1 -2925.764,E2 -2925.764} C_VEL
LIN {X 0,Y 559.174,Z 280.83,A -85,B 0,C 180,E1 -2928.237,E2 -2928.237} C_VEL
LIN {X 0,Y 559.156,Z 280.83,A -85,B 0,C 180,E1 -2931.194,E2 -2931.194} C_VEL
LIN {X 0,Y 559.151,Z 280.838,A -85,B 0,C 180,E1 -2933.796,E2 -2933.796} C_VEL
LIN {X 0,Y 559.158,Z 280.832,A -85,B 0,C 180,E1 -2936.43,E2 -2936.43} C_VEL
LIN {X 0,Y 559.151,Z 280.831,A -85,B 0,C 180,E1 -2938.986,E2 -2938.986} C_VEL
LIN {X 0,Y 559.156,Z 280.834,A -85,B 0,C 180,E1 -2941.622,E2 -2941.622} C_VEL
LIN {X 0,Y 559.187,Z 280.834,A -85,B 0,C 180,E1 -2943.908,E2 -2943.908} C_VEL
LIN {X 0,Y 559.211,Z 280.928,A -85,B 0,C 180,E1 -2946.291,E2 -2946.291} C_VEL
LIN {X 0,Y 560.08,Z 286.299,A -85,B 0,C 180,E1 -2947.112,E2 -2947.112} C_VEL
LIN {X 0,Y 559.865,Z 308.311,A -85,B 0,C 180,E1 -2950.302,E2 -2950.302} C_VEL
LIN {X 0,Y 559.593,Z 328.677,A -85,B 0,C 180,E1 -2953.214,E2 -2953.214} C_VEL
LIN {X 0,Y 559.403,Z 346.718,A -85,B 0,C 180,E1 -2955.811,E2 -2955.811} C_VEL
LIN {X 0,Y 560.298,Z 353.502,A -85,B 0,C 180,E1 -2955.924,E2 -2955.924} C_VEL
LIN {X 0,Y 560.019,Z 455.109,A -85,B 0,C 180,E1 -2957.248,E2 -2957.248} C_VEL
LIN {X 0,Y 559.882,Z 468.326,A -85,B 0,C 180,E1 -2957.567,E2 -2957.567} C_VEL
LIN {X 0,Y 559.77,Z 480.457,A -85,B 0,C 180,E1 -2958.002,E2 -2958.002} C_VEL
LIN {X 0,Y 559.663,Z 491.869,A -85,B 0,C 180,E1 -2958.55,E2 -2958.55} C_VEL
LIN {X 0,Y 559.503,Z 502.949,A -85,B 0,C 180,E1 -2959.234,E2 -2959.234} C_VEL
LIN {X 0,Y 559.307,Z 513.574,A -85,B 0,C 180,E1 -2960.054,E2 -2960.054} C_VEL
LIN {X 0,Y 559.159,Z 523.125,A -85,B 0,C 180,E1 -2960.964,E2 -2960.964} C_VEL
LIN {X 0,Y 559.047,Z 530.984,A -85,B 0,C 180,E1 -2961.872,E2 -2961.872} C_VEL
LIN {X 0,Y 558.948,Z 538.64,A -85,B 0,C 180,E1 -2962.961,E2 -2962.961} C_VEL
LIN {X 0,Y 558.938,Z 545.693,A -85,B 0,C 180,E1 -2964.23,E2 -2964.23} C_VEL
LIN {X 0,Y 558.826,Z 550.383,A -85,B 0,C 180,E1 -2965.314,E2 -2965.314} C_VEL
LIN {X 0,Y 558.835,Z 553.966,A -85,B 0,C 180,E1 -2966.397,E2 -2966.397} C_VEL
LIN {X 0,Y 558.799,Z 555.813,A -85,B 0,C 180,E1 -2967.119,E2 -2967.119} C_VEL
LIN {X 0,Y 558.745,Z 558.187,A -85,B 0,C 180,E1 -2968.561,E2 -2968.561} C_VEL
LIN {X 0,Y 558.74,Z 559,A -85,B 0,C 180,E1 -2970.002,E2 -2970.002} C_VEL
LIN {X 0,Y 558.745,Z 558.182,A -85,B 0,C 180,E1 -2971.444,E2 -2971.444} C_VEL
LIN {X 0,Y 558.799,Z 555.805,A -85,B 0,C 180,E1 -2972.886,E2 -2972.886} C_VEL
LIN {X 0,Y 558.844,Z 552.889,A -85,B 0,C 180,E1 -2973.968,E2 -2973.968} C_VEL
LIN {X 0,Y 558.798,Z 548.941,A -85,B 0,C 180,E1 -2975.053,E2 -2975.053} C_VEL
LIN {X 0,Y 558.926,Z 543.857,A -85,B 0,C 180,E1 -2976.137,E2 -2976.137} C_VEL
LIN {X 0,Y 558.979,Z 537.455,A -85,B 0,C 180,E1 -2977.225,E2 -2977.225} C_VEL
LIN {X 0,Y 559.093,Z 529.463,A -85,B 0,C 180,E1 -2978.314,E2 -2978.314} C_VEL
LIN {X 0,Y 559.186,Z 521.317,A -85,B 0,C 180,E1 -2979.223,E2 -2979.223} C_VEL
LIN {X 0,Y 559.338,Z 511.379,A -85,B 0,C 180,E1 -2980.133,E2 -2980.133} C_VEL
LIN {X 0,Y 559.57,Z 500.36,A -85,B 0,C 180,E1 -2980.939,E2 -2980.939} C_VEL
LIN {X 0,Y 559.675,Z 488.429,A -85,B 0,C 180,E1 -2981.629,E2 -2981.629} C_VEL
LIN {X 0,Y 559.816,Z 475.724,A -85,B 0,C 180,E1 -2982.186,E2 -2982.186} C_VEL
LIN {X 0,Y 559.927,Z 462.285,A -85,B 0,C 180,E1 -2982.598,E2 -2982.598} C_VEL
LIN {X 0,Y 560.049,Z 448.977,A -85,B 0,C 180,E1 -2982.849,E2 -2982.849} C_VEL
LIN {X 0,Y 560.2,Z 352.174,A -85,B 0,C 180,E1 -2984.095,E2 -2984.095} C_VEL
LIN {X 0,Y 559.393,Z 346.603,A -85,B 0,C 180,E1 -2984.206,E2 -2984.206} C_VEL
LIN {X 0,Y 559.627,Z 326.675,A -85,B 0,C 180,E1 -2987.075,E2 -2987.075} C_VEL
LIN {X 0,Y 559.891,Z 306.358,A -85,B 0,C 180,E1 -2990.003,E2 -2990.003} C_VEL
LIN {X 0,Y 560.149,Z 287.948,A -85,B 0,C 180,E1 -2992.695,E2 -2992.695} C_VEL
LIN {X 0,Y 559.631,Z 283.41,A -85,B 0,C 180,E1 -2993.393,E2 -2993.393} C_VEL
LIN {X 0,Y 559.162,Z 280.837,A -85,B 0,C 180,E1 -2993.815,E2 -2993.815} C_VEL
LIN {X 0,Y 559.18,Z 280.835,A -85,B 0,C 180,E1 -2996.098,E2 -2996.098} C_VEL
LIN {X 0,Y 559.144,Z 280.833,A -85,B 0,C 180,E1 -2998.531,E2 -2998.531} C_VEL
LIN {X 0,Y 559.149,Z 280.83,A -85,B 0,C 180,E1 -3001.273,E2 -3001.273} C_VEL
LIN {X 0,Y 559.168,Z 280.833,A -85,B 0,C 180,E1 -3003.949,E2 -3003.949} C_VEL
LIN {X 0,Y 559.142,Z 280.83,A -85,B 0,C 180,E1 -3007.108,E2 -3007.108} C_VEL
LIN {X 0,Y 559.16,Z 280.832,A -85,B 0,C 180,E1 -3009.941,E2 -3009.941} C_VEL
LIN {X 0,Y 559.16,Z 280.831,A -85,B 0,C 180,E1 -3012.743,E2 -3012.743} C_VEL
LIN {X 0,Y 559.146,Z 280.83,A -85,B 0,C 180,E1 -3015.761,E2 -3015.761} C_VEL
LIN {X 0,Y 559.188,Z 280.83,A -85,B 0,C 180,E1 -3018.232,E2 -3018.232} C_VEL
LIN {X 0,Y 559.173,Z 280.827,A -85,B 0,C 180,E1 -3021.191,E2 -3021.191} C_VEL
LIN {X 0,Y 559.155,Z 280.828,A -85,B 0,C 180,E1 -3023.79,E2 -3023.79} C_VEL
LIN {X 0,Y 559.158,Z 280.833,A -85,B 0,C 180,E1 -3026.425,E2 -3026.425} C_VEL
LIN {X 0,Y 559.159,Z 280.834,A -85,B 0,C 180,E1 -3028.981,E2 -3028.981} C_VEL
LIN {X 0,Y 559.16,Z 280.828,A -85,B 0,C 180,E1 -3031.618,E2 -3031.618} C_VEL
LIN {X 0,Y 559.19,Z 280.823,A -85,B 0,C 180,E1 -3033.903,E2 -3033.903} C_VEL
LIN {X 0,Y 559.147,Z 280.833,A -85,B 0,C 180,E1 -3036.567,E2 -3036.567} C_VEL
LIN {X 0,Y 559.167,Z 280.83,A -85,B 0,C 180,E1 -3039.395,E2 -3039.395} C_VEL
LIN {X 0,Y 559.134,Z 280.832,A -85,B 0,C 180,E1 -3041.685,E2 -3041.685} C_VEL
LIN {X 0,Y 559.153,Z 280.828,A -85,B 0,C 180,E1 -3043.947,E2 -3043.947} C_VEL
LIN {X 0,Y 559.16,Z 280.827,A -85,B 0,C 180,E1 -3046.184,E2 -3046.184} C_VEL
LIN {X 0,Y 559.188,Z 280.833,A -85,B 0,C 180,E1 -3049.133,E2 -3049.133} C_VEL
LIN {X 0,Y 559.188,Z 280.824,A -85,B 0,C 180,E1 -3052.053,E2 -3052.053} C_VEL
LIN {X 0,Y 559.247,Z 280.82,A -85,B 0,C 180,E1 -3054.953,E2 -3054.953} C_VEL
LIN {X 0,Y 559.23,Z 280.822,A -85,B 0,C 180,E1 -3057.839,E2 -3057.839} C_VEL
LIN {X 0,Y 559.236,Z 280.82,A -85,B 0,C 180,E1 -3060,E2 -3060} C_VEL
LIN {X 0,Y 559.222,Z 280.82,A -85,B 0,C 180,E1 -3062.881,E2 -3062.881} C_VEL
LIN {X 0,Y 559.209,Z 280.829,A -85,B 0,C 180,E1 -3065.77,E2 -3065.77} C_VEL
LIN {X 0,Y 559.154,Z 280.828,A -85,B 0,C 180,E1 -3068.675,E2 -3068.675} C_VEL
LIN {X 0,Y 559.191,Z 280.831,A -85,B 0,C 180,E1 -3071.601,E2 -3071.601} C_VEL
LIN {X 0,Y 559.168,Z 280.827,A -85,B 0,C 180,E1 -3074.588,E2 -3074.588} C_VEL
LIN {X 0,Y 559.126,Z 280.836,A -85,B 0,C 180,E1 -3077.558,E2 -3077.558} C_VEL
LIN {X 0,Y 559.15,Z 280.837,A -85,B 0,C 180,E1 -3079.838,E2 -3079.838} C_VEL
LIN {X 0,Y 559.121,Z 280.84,A -85,B 0,C 180,E1 -3082.154,E2 -3082.154} C_VEL
LIN {X 0,Y 559.13,Z 280.831,A -85,B 0,C 180,E1 -3085.179,E2 -3085.179} C_VEL
LIN {X 0,Y 559.095,Z 280.839,A -85,B 0,C 180,E1 -3087.717,E2 -3087.717} C_VEL
LIN {X 0,Y 559.119,Z 280.836,A -85,B 0,C 180,E1 -3090.594,E2 -3090.594} C_VEL
LIN {X 0,Y 558.463,Z 280.916,A -85,B 0,C 180,E1 -3091.196,E2 -3091.196} C_VEL
LIN {X 0,Y 555.604,Z 281.279,A -85,B 0,C 180,E1 -3092.172,E2 -3092.172} C_VEL
LIN {X 0,Y 553.186,Z 281.575,A -85,B 0,C 180,E1 -3092.958,E2 -3092.958} C_VEL
LIN {X 0,Y 552.156,Z 281.701,A -85,B 0,C 180,E1 -3093.565,E2 -3093.565} C_VEL
LIN {X 0,Y 552.078,Z 281.712,A -85,B 0,C 180,E1 -3093.77,E2 -3093.77} C_VEL
LIN {X 0,Y 552.045,Z 281.718,A -85,B 0,C 180,E1 -3096.752,E2 -3096.752} C_VEL
LIN {X 0,Y 552.075,Z 281.71,A -85,B 0,C 180,E1 -3099.532,E2 -3099.532} C_VEL
LIN {X 0,Y 552.075,Z 281.719,A -85,B 0,C 180,E1 -3102.431,E2 -3102.431} C_VEL
LIN {X 0,Y 552.061,Z 281.711,A -85,B 0,C 180,E1 -3105.559,E2 -3105.559} C_VEL
LIN {X 0,Y 552.048,Z 281.722,A -85,B 0,C 180,E1 -3108.548,E2 -3108.548} C_VEL
LIN {X 0,Y 552.056,Z 281.713,A -85,B 0,C 180,E1 -3111.406,E2 -3111.406} C_VEL
LIN {X 0,Y 552.048,Z 281.715,A -85,B 0,C 180,E1 -3114.153,E2 -3114.153} C_VEL
LIN {X 0,Y 552.087,Z 281.713,A -85,B 0,C 180,E1 -3117.159,E2 -3117.159} C_VEL
LIN {X 0,Y 552.059,Z 281.712,A -85,B 0,C 180,E1 -3119.96,E2 -3119.96} C_VEL
LIN {X 0,Y 552.065,Z 281.717,A -85,B 0,C 180,E1 -3122.722,E2 -3122.722} C_VEL
LIN {X 0,Y 552.049,Z 281.721,A -85,B 0,C 180,E1 -3125.157,E2 -3125.157} C_VEL
LIN {X 0,Y 552.082,Z 281.712,A -85,B 0,C 180,E1 -3127.548,E2 -3127.548} C_VEL
LIN {X 0,Y 552.125,Z 281.704,A -85,B 0,C 180,E1 -3130.382,E2 -3130.382} C_VEL
LIN {X 0,Y 552.111,Z 281.711,A -85,B 0,C 180,E1 -3132.975,E2 -3132.975} C_VEL
LIN {X 0,Y 552.117,Z 281.705,A -85,B 0,C 180,E1 -3136.003,E2 -3136.003} C_VEL
LIN {X 0,Y 552.157,Z 281.704,A -85,B 0,C 180,E1 -3138.992,E2 -3138.992} C_VEL
LIN {X 0,Y 552.111,Z 281.708,A -85,B 0,C 180,E1 -3141.949,E2 -3141.949} C_VEL
LIN {X 0,Y 552.215,Z 281.694,A -85,B 0,C 180,E1 -3144.887,E2 -3144.887} C_VEL
LIN {X 0,Y 552.221,Z 281.698,A -85,B 0,C 180,E1 -3147.81,E2 -3147.81} C_VEL
LIN {X 0,Y 552.225,Z 281.695,A -85,B 0,C 180,E1 -3149.998,E2 -3149.998} C_VEL
LIN {X 0,Y 552.183,Z 281.697,A -85,B 0,C 180,E1 -3152.916,E2 -3152.916} C_VEL
LIN {X 0,Y 552.184,Z 281.707,A -85,B 0,C 180,E1 -3155.841,E2 -3155.841} C_VEL
LIN {X 0,Y 552.136,Z 281.704,A -85,B 0,C 180,E1 -3158.783,E2 -3158.783} C_VEL
LIN {X 0,Y 552.141,Z 281.712,A -85,B 0,C 180,E1 -3161.748,E2 -3161.748} C_VEL
LIN {X 0,Y 552.162,Z 281.877,A -85,B 0,C 180,E1 -3162.727,E2 -3162.727} C_VEL
LIN {X 0,Y 552.43,Z 288.557,A -85,B 0,C 180,E1 -3163.984,E2 -3163.984} C_VEL
LIN {X 0,Y 552.262,Z 302.832,A -85,B 0,C 180,E1 -3166.635,E2 -3166.635} C_VEL
LIN {X 0,Y 552.204,Z 308.444,A -85,B 0,C 180,E1 -3167.679,E2 -3167.679} C_VEL
LIN {X 0,Y 553.38,Z 315.41,A -85,B 0,C 180,E1 -3167.814,E2 -3167.814} C_VEL
LIN {X 0,Y 553.1,Z 414.514,A -85,B 0,C 180,E1 -3169.119,E2 -3169.119} C_VEL
LIN {X 0,Y 552.998,Z 428.083,A -85,B 0,C 180,E1 -3169.447,E2 -3169.447} C_VEL
LIN {X 0,Y 552.849,Z 440.52,A -85,B 0,C 180,E1 -3169.897,E2 -3169.897} C_VEL
LIN {X 0,Y 552.63,Z 452.213,A -85,B 0,C 180,E1 -3170.467,E2 -3170.467} C_VEL
LIN {X 0,Y 552.436,Z 463.178,A -85,B 0,C 180,E1 -3171.156,E2 -3171.156} C_VEL
LIN {X 0,Y 552.292,Z 473.962,A -85,B 0,C 180,E1 -3172.005,E2 -3172.005} C_VEL
LIN {X 0,Y 552.122,Z 482.642,A -85,B 0,C 180,E1 -3172.841,E2 -3172.841} C_VEL
LIN {X 0,Y 551.976,Z 491.658,A -85,B 0,C 180,E1 -3173.902,E2 -3173.902} C_VEL
LIN {X 0,Y 551.865,Z 499.544,A -85,B 0,C 180,E1 -3175.064,E2 -3175.064} C_VEL
LIN {X 0,Y 551.802,Z 505.011,A -85,B 0,C 180,E1 -3176.061,E2 -3176.061} C_VEL
LIN {X 0,Y 551.734,Z 510.35,A -85,B 0,C 180,E1 -3177.29,E2 -3177.29} C_VEL
LIN {X 0,Y 551.708,Z 514.217,A -85,B 0,C 180,E1 -3178.482,E2 -3178.482} C_VEL
LIN {X 0,Y 551.677,Z 517.375,A -85,B 0,C 180,E1 -3179.971,E2 -3179.971} C_VEL
LIN {X 0,Y 551.64,Z 518.837,A -85,B 0,C 180,E1 -3181.395,E2 -3181.395} C_VEL
LIN {X 0,Y 551.662,Z 518.787,A -85,B 0,C 180,E1 -3182.773,E2 -3182.773} C_VEL
LIN {X 0,Y 551.668,Z 517.404,A -85,B 0,C 180,E1 -3184.099,E2 -3184.099} C_VEL
LIN {X 0,Y 551.692,Z 514.797,A -85,B 0,C 180,E1 -3185.383,E2 -3185.383} C_VEL
LIN {X 0,Y 551.756,Z 510.474,A -85,B 0,C 180,E1 -3186.768,E2 -3186.768} C_VEL
LIN {X 0,Y 551.772,Z 505.934,A -85,B 0,C 180,E1 -3187.842,E2 -3187.842} C_VEL
LIN {X 0,Y 551.875,Z 499.521,A -85,B 0,C 180,E1 -3189.029,E2 -3189.029} C_VEL
LIN {X 0,Y 551.997,Z 491.649,A -85,B 0,C 180,E1 -3190.189,E2 -3190.189} C_VEL
LIN {X 0,Y 552.113,Z 483.66,A -85,B 0,C 180,E1 -3191.141,E2 -3191.141} C_VEL
LIN {X 0,Y 552.285,Z 474.544,A -85,B 0,C 180,E1 -3192.035,E2 -3192.035} C_VEL
LIN {X 0,Y 552.418,Z 464.525,A -85,B 0,C 180,E1 -3192.837,E2 -3192.837} C_VEL
LIN {X 0,Y 552.596,Z 453.707,A -85,B 0,C 180,E1 -3193.536,E2 -3193.536} C_VEL
LIN {X 0,Y 552.809,Z 442.015,A -85,B 0,C 180,E1 -3194.13,E2 -3194.13} C_VEL
LIN {X 0,Y 552.996,Z 429.362,A -85,B 0,C 180,E1 -3194.604,E2 -3194.604} C_VEL
LIN {X 0,Y 553.101,Z 415.946,A -85,B 0,C 180,E1 -3194.942,E2 -3194.942} C_VEL
LIN {X 0,Y 553.309,Z 356.833,A -85,B 0,C 180,E1 -3195.735,E2 -3195.735} C_VEL
LIN {X 0,Y 553.362,Z 315.413,A -85,B 0,C 180,E1 -3196.276,E2 -3196.276} C_VEL
LIN {X 0,Y 552.202,Z 308.43,A -85,B 0,C 180,E1 -3196.407,E2 -3196.407} C_VEL
LIN {X 0,Y 552.316,Z 295.985,A -85,B 0,C 180,E1 -3198.647,E2 -3198.647} C_VEL
LIN {X 0,Y 552.326,Z 285.443,A -85,B 0,C 180,E1 -3200.489,E2 -3200.489} C_VEL
LIN {X 0,Y 552.15,Z 281.707,A -85,B 0,C 180,E1 -3201.158,E2 -3201.158} C_VEL
LIN {X 0,Y 552.074,Z 281.72,A -85,B 0,C 180,E1 -3204.155,E2 -3204.155} C_VEL
LIN {X 0,Y 552.087,Z 281.712,A -85,B 0,C 180,E1 -3206.812,E2 -3206.812} C_VEL
LIN {X 0,Y 552.071,Z 281.712,A -85,B 0,C 180,E1 -3209.389,E2 -3209.389} C_VEL
LIN {X 0,Y 552.08,Z 281.714,A -85,B 0,C 180,E1 -3211.9,E2 -3211.9} C_VEL
LIN {X 0,Y 552.114,Z 281.713,A -85,B 0,C 180,E1 -3214.645,E2 -3214.645} C_VEL
LIN {X 0,Y 552.047,Z 281.716,A -85,B 0,C 180,E1 -3217.547,E2 -3217.547} C_VEL
LIN {X 0,Y 552.103,Z 281.715,A -85,B 0,C 180,E1 -3220.672,E2 -3220.672} C_VEL
LIN {X 0,Y 552.064,Z 281.712,A -85,B 0,C 180,E1 -3223.736,E2 -3223.736} C_VEL
LIN {X 0,Y 552.083,Z 281.711,A -85,B 0,C 180,E1 -3226.003,E2 -3226.003} C_VEL
LIN {X 0,Y 552.125,Z 281.708,A -85,B 0,C 180,E1 -3228.993,E2 -3228.993} C_VEL
LIN {X 0,Y 552.106,Z 281.707,A -85,B 0,C 180,E1 -3231.951,E2 -3231.951} C_VEL
LIN {X 0,Y 552.179,Z 281.705,A -85,B 0,C 180,E1 -3234.888,E2 -3234.888} C_VEL
LIN {X 0,Y 552.161,Z 281.699,A -85,B 0,C 180,E1 -3237.812,E2 -3237.812} C_VEL
LIN {X 0,Y 552.2,Z 281.701,A -85,B 0,C 180,E1 -3240.729,E2 -3240.729} C_VEL
LIN {X 0,Y 552.164,Z 281.708,A -85,B 0,C 180,E1 -3242.918,E2 -3242.918} C_VEL
LIN {X 0,Y 552.153,Z 281.701,A -85,B 0,C 180,E1 -3245.844,E2 -3245.844} C_VEL
LIN {X 0,Y 552.124,Z 281.709,A -85,B 0,C 180,E1 -3248.786,E2 -3248.786} C_VEL
LIN {X 0,Y 552.113,Z 281.705,A -85,B 0,C 180,E1 -3251.752,E2 -3251.752} C_VEL
LIN {X 0,Y 552.085,Z 281.713,A -85,B 0,C 180,E1 -3254.75,E2 -3254.75} C_VEL
LIN {X 0,Y 552.085,Z 281.71,A -85,B 0,C 180,E1 -3257.789,E2 -3257.789} C_VEL
LIN {X 0,Y 552.086,Z 281.707,A -85,B 0,C 180,E1 -3260.103,E2 -3260.103} C_VEL
LIN {X 0,Y 552.107,Z 281.706,A -85,B 0,C 180,E1 -3262.45,E2 -3262.45} C_VEL
LIN {X 0,Y 552.135,Z 281.711,A -85,B 0,C 180,E1 -3265.36,E2 -3265.36} C_VEL
LIN {X 0,Y 552.095,Z 281.707,A -85,B 0,C 180,E1 -3268.099,E2 -3268.099} C_VEL
LIN {X 0,Y 552.074,Z 281.71,A -85,B 0,C 180,E1 -3270.611,E2 -3270.611} C_VEL
LIN {X 0,Y 552.095,Z 281.712,A -85,B 0,C 180,E1 -3273.187,E2 -3273.187} C_VEL
LIN {X 0,Y 552.082,Z 281.715,A -85,B 0,C 180,E1 -3275.844,E2 -3275.844} C_VEL
LIN {X 0,Y 552.095,Z 281.707,A -85,B 0,C 180,E1 -3278.591,E2 -3278.591} C_VEL
LIN {X 0,Y 552.141,Z 281.709,A -85,B 0,C 180,E1 -3281.444,E2 -3281.444} C_VEL
LIN {X 0,Y 552.064,Z 281.713,A -85,B 0,C 180,E1 -3284.536,E2 -3284.536} C_VEL
LIN {X 0,Y 552.102,Z 281.716,A -85,B 0,C 180,E1 -3287.588,E2 -3287.588} C_VEL
LIN {X 0,Y 552.117,Z 281.715,A -85,B 0,C 180,E1 -3289.796,E2 -3289.796} C_VEL
LIN {X 0,Y 552.072,Z 281.714,A -85,B 0,C 180,E1 -3292.341,E2 -3292.341} C_VEL
LIN {X 0,Y 552.11,Z 281.707,A -85,B 0,C 180,E1 -3295.059,E2 -3295.059} C_VEL
LIN {X 0,Y 552.11,Z 281.714,A -85,B 0,C 180,E1 -3297.686,E2 -3297.686} C_VEL
LIN {X 0,Y 552.129,Z 281.712,A -85,B 0,C 180,E1 -3300.241,E2 -3300.241} C_VEL
LIN {X 0,Y 552.134,Z 281.705,A -85,B 0,C 180,E1 -3303.002,E2 -3303.002} C_VEL
LIN {X 0,Y 552.169,Z 281.709,A -85,B 0,C 180,E1 -3306.091,E2 -3306.091} C_VEL
LIN {X 0,Y 552.167,Z 281.786,A -85,B 0,C 180,E1 -3306.151,E2 -3306.151} C_VEL
LIN {X 0,Y 553.172,Z 288.624,A -85,B 0,C 180,E1 -3307.205,E2 -3307.205} C_VEL
LIN {X 0,Y 552.856,Z 310.625,A -85,B 0,C 180,E1 -3310.433,E2 -3310.433} C_VEL
LIN {X 0,Y 552.557,Z 329.666,A -85,B 0,C 180,E1 -3313.184,E2 -3313.184} C_VEL
LIN {X 0,Y 552.367,Z 346.728,A -85,B 0,C 180,E1 -3315.628,E2 -3315.628} C_VEL
LIN {X 0,Y 553.411,Z 355.023,A -85,B 0,C 180,E1 -3315.766,E2 -3315.766} C_VEL
LIN {X 0,Y 553.106,Z 455.109,A -85,B 0,C 180,E1 -3317.086,E2 -3317.086} C_VEL
LIN {X 0,Y 552.962,Z 468.325,A -85,B 0,C 180,E1 -3317.409,E2 -3317.409} C_VEL
LIN {X 0,Y 552.817,Z 481.236,A -85,B 0,C 180,E1 -3317.881,E2 -3317.881} C_VEL
LIN {X 0,Y 552.678,Z 493.681,A -85,B 0,C 180,E1 -3318.509,E2 -3318.509} C_VEL
LIN {X 0,Y 552.464,Z 505.529,A -85,B 0,C 180,E1 -3319.281,E2 -3319.281} C_VEL
LIN {X 0,Y 552.274,Z 515.679,A -85,B 0,C 180,E1 -3320.111,E2 -3320.111} C_VEL
LIN {X 0,Y 552.103,Z 524.812,A -85,B 0,C 180,E1 -3321.032,E2 -3321.032} C_VEL
LIN {X 0,Y 551.957,Z 533.71,A -85,B 0,C 180,E1 -3322.136,E2 -3322.136} C_VEL
LIN {X 0,Y 551.889,Z 539.757,A -85,B 0,C 180,E1 -3323.055,E2 -3323.055} C_VEL
LIN {X 0,Y 551.87,Z 545.693,A -85,B 0,C 180,E1 -3324.155,E2 -3324.155} C_VEL
LIN {X 0,Y 551.724,Z 550.383,A -85,B 0,C 180,E1 -3325.253,E2 -3325.253} C_VEL
LIN {X 0,Y 551.75,Z 553.966,A -85,B 0,C 180,E1 -3326.351,E2 -3326.351} C_VEL
LIN {X 0,Y 551.723,Z 555.813,A -85,B 0,C 180,E1 -3327.082,E2 -3327.082} C_VEL
LIN {X 0,Y 551.645,Z 558.186,A -85,B 0,C 180,E1 -3328.542,E2 -3328.542} C_VEL
LIN {X 0,Y 551.64,Z 559,A -85,B 0,C 180,E1 -3330.002,E2 -3330.002} C_VEL
LIN {X 0,Y 551.645,Z 558.182,A -85,B 0,C 180,E1 -3331.462,E2 -3331.462} C_VEL
LIN {X 0,Y 551.724,Z 555.805,A -85,B 0,C 180,E1 -3332.923,E2 -3332.923} C_VEL
LIN {X 0,Y 551.764,Z 552.889,A -85,B 0,C 180,E1 -3334.019,E2 -3334.019} C_VEL
LIN {X 0,Y 551.724,Z 548.94,A -85,B 0,C 180,E1 -3335.118,E2 -3335.118} C_VEL
LIN {X 0,Y 551.828,Z 543.175,A -85,B 0,C 180,E1 -3336.344,E2 -3336.344} C_VEL
LIN {X 0,Y 551.928,Z 536.223,A -85,B 0,C 180,E1 -3337.501,E2 -3337.501} C_VEL
LIN {X 0,Y 552.065,Z 527.977,A -85,B 0,C 180,E1 -3338.604,E2 -3338.604} C_VEL
LIN {X 0,Y 552.224,Z 519.522,A -85,B 0,C 180,E1 -3339.525,E2 -3339.525} C_VEL
LIN {X 0,Y 552.382,Z 509.071,A -85,B 0,C 180,E1 -3340.447,E2 -3340.447} C_VEL
LIN {X 0,Y 552.615,Z 498.227,A -85,B 0,C 180,E1 -3341.217,E2 -3341.217} C_VEL
LIN {X 0,Y 552.753,Z 487.374,A -85,B 0,C 180,E1 -3341.832,E2 -3341.832} C_VEL
LIN {X 0,Y 552.881,Z 475.72,A -85,B 0,C 180,E1 -3342.342,E2 -3342.342} C_VEL
LIN {X 0,Y 553.017,Z 462.284,A -85,B 0,C 180,E1 -3342.758,E2 -3342.758} C_VEL
LIN {X 0,Y 553.143,Z 448.977,A -85,B 0,C 180,E1 -3343.012,E2 -3343.012} C_VEL
LIN {X 0,Y 553.326,Z 352.871,A -85,B 0,C 180,E1 -3344.265,E2 -3344.265} C_VEL
LIN {X 0,Y 552.389,Z 346.568,A -85,B 0,C 180,E1 -3344.394,E2 -3344.394} C_VEL
LIN {X 0,Y 552.637,Z 325.159,A -85,B 0,C 180,E1 -3347.485,E2 -3347.485} C_VEL
LIN {X 0,Y 552.939,Z 304.814,A -85,B 0,C 180,E1 -3350.46,E2 -3350.46} C_VEL
LIN {X 0,Y 553.192,Z 287.74,A -85,B 0,C 180,E1 -3352.997,E2 -3352.997} C_VEL
LIN {X 0,Y 552.144,Z 281.71,A -85,B 0,C 180,E1 -3353.978,E2 -3353.978} C_VEL
LIN {X 0,Y 552.138,Z 281.704,A -85,B 0,C 180,E1 -3356.999,E2 -3356.999} C_VEL
LIN {X 0,Y 552.12,Z 281.715,A -85,B 0,C 180,E1 -3360.051,E2 -3360.051} C_VEL
LIN {X 0,Y 552.117,Z 281.705,A -85,B 0,C 180,E1 -3362.846,E2 -3362.846} C_VEL
LIN {X 0,Y 552.078,Z 281.71,A -85,B 0,C 180,E1 -3365.439,E2 -3365.439} C_VEL
LIN {X 0,Y 552.097,Z 281.711,A -85,B 0,C 180,E1 -3367.885,E2 -3367.885} C_VEL
LIN {X 0,Y 552.11,Z 281.713,A -85,B 0,C 180,E1 -3370.481,E2 -3370.481} C_VEL
LIN {X 0,Y 552.106,Z 281.706,A -85,B 0,C 180,E1 -3373.423,E2 -3373.423} C_VEL
LIN {X 0,Y 552.104,Z 281.715,A -85,B 0,C 180,E1 -3376.576,E2 -3376.576} C_VEL
LIN {X 0,Y 552.117,Z 281.704,A -85,B 0,C 180,E1 -3379.519,E2 -3379.519} C_VEL
LIN {X 0,Y 552.089,Z 281.714,A -85,B 0,C 180,E1 -3382.336,E2 -3382.336} C_VEL
LIN {X 0,Y 552.113,Z 281.709,A -85,B 0,C 180,E1 -3385.053,E2 -3385.053} C_VEL
LIN {X 0,Y 552.121,Z 281.704,A -85,B 0,C 180,E1 -3387.682,E2 -3387.682} C_VEL
LIN {X 0,Y 552.137,Z 281.704,A -85,B 0,C 180,E1 -3390.236,E2 -3390.236} C_VEL
LIN {X 0,Y 552.138,Z 281.71,A -85,B 0,C 180,E1 -3392.998,E2 -3392.998} C_VEL
LIN {X 0,Y 552.104,Z 281.712,A -85,B 0,C 180,E1 -3395.161,E2 -3395.161} C_VEL
LIN {X 0,Y 552.085,Z 281.71,A -85,B 0,C 180,E1 -3397.549,E2 -3397.549} C_VEL
LIN {X 0,Y 552.144,Z 281.706,A -85,B 0,C 180,E1 -3400.674,E2 -3400.674} C_VEL
LIN {X 0,Y 552.103,Z 281.708,A -85,B 0,C 180,E1 -3403.737,E2 -3403.737} C_VEL
LIN {X 0,Y 552.123,Z 281.704,A -85,B 0,C 180,E1 -3406.004,E2 -3406.004} C_VEL
LIN {X 0,Y 552.155,Z 281.706,A -85,B 0,C 180,E1 -3408.993,E2 -3408.993} C_VEL
LIN {X 0,Y 552.142,Z 281.703,A -85,B 0,C 180,E1 -3411.951,E2 -3411.951} C_VEL
LIN {X 0,Y 552.221,Z 281.695,A -85,B 0,C 180,E1 -3414.889,E2 -3414.889} C_VEL
LIN {X 0,Y 552.203,Z 281.698,A -85,B 0,C 180,E1 -3417.812,E2 -3417.812} C_VEL
LIN {X 0,Y 552.226,Z 281.691,A -85,B 0,C 180,E1 -3420.729,E2 -3420.729} C_VEL
LIN {X 0,Y 552.19,Z 281.697,A -85,B 0,C 180,E1 -3422.918,E2 -3422.918} C_VEL
LIN {X 0,Y 552.177,Z 281.704,A -85,B 0,C 180,E1 -3425.844,E2 -3425.844} C_VEL
LIN {X 0,Y 552.13,Z 281.703,A -85,B 0,C 180,E1 -3428.786,E2 -3428.786} C_VEL
LIN {X 0,Y 552.148,Z 281.711,A -85,B 0,C 180,E1 -3431.751,E2 -3431.751} C_VEL
LIN {X 0,Y 552.115,Z 281.705,A -85,B 0,C 180,E1 -3434.749,E2 -3434.749} C_VEL
LIN {X 0,Y 552.085,Z 281.717,A -85,B 0,C 180,E1 -3437.789,E2 -3437.789} C_VEL
LIN {X 0,Y 552.112,Z 281.713,A -85,B 0,C 180,E1 -3440.102,E2 -3440.102} C_VEL
LIN {X 0,Y 552.073,Z 281.713,A -85,B 0,C 180,E1 -3442.452,E2 -3442.452} C_VEL
LIN {X 0,Y 552.074,Z 281.71,A -85,B 0,C 180,E1 -3445.335,E2 -3445.335} C_VEL
LIN {X 0,Y 552.045,Z 281.723,A -85,B 0,C 180,E1 -3448.102,E2 -3448.102} C_VEL
LIN {X 0,Y 552.084,Z 281.713,A -85,B 0,C 180,E1 -3450.611,E2 -3450.611} C_VEL
LIN {X 0,Y 552.097,Z 281.707,A -85,B 0,C 180,E1 -3453.187,E2 -3453.187} C_VEL
LIN {X 0,Y 552.078,Z 281.712,A -85,B 0,C 180,E1 -3453.77,E2 -3453.77} C_VEL
LIN {X 0,Y 551.419,Z 281.801,A -85,B 0,C 180,E1 -3454.379,E2 -3454.379} C_VEL
LIN {X 0,Y 548.547,Z 282.16,A -85,B 0,C 180,E1 -3455.367,E2 -3455.367} C_VEL
LIN {X 0,Y 546.116,Z 282.46,A -85,B 0,C 180,E1 -3456.162,E2 -3456.162} C_VEL
LIN {X 0,Y 545.076,Z 282.586,A -85,B 0,C 180,E1 -3456.776,E2 -3456.776} C_VEL
LIN {X 0,Y 544.994,Z 282.593,A -85,B 0,C 180,E1 -3456.984,E2 -3456.984} C_VEL
LIN {X 0,Y 545.031,Z 282.587,A -85,B 0,C 180,E1 -3459.315,E2 -3459.315} C_VEL
LIN {X 0,Y 545.023,Z 282.592,A -85,B 0,C 180,E1 -3462.108,E2 -3462.108} C_VEL
LIN {X 0,Y 545.01,Z 282.591,A -85,B 0,C 180,E1 -3465.173,E2 -3465.173} C_VEL
LIN {X 0,Y 545.017,Z 282.595,A -85,B 0,C 180,E1 -3468.41,E2 -3468.41} C_VEL
LIN {X 0,Y 545.02,Z 282.597,A -85,B 0,C 180,E1 -3470.813,E2 -3470.813} C_VEL
LIN {X 0,Y 544.994,Z 282.592,A -85,B 0,C 180,E1 -3473.616,E2 -3473.616} C_VEL
LIN {X 0,Y 545.037,Z 282.595,A -85,B 0,C 180,E1 -3476.945,E2 -3476.945} C_VEL
LIN {X 0,Y 545.01,Z 282.59,A -85,B 0,C 180,E1 -3479.807,E2 -3479.807} C_VEL
LIN {X 0,Y 544.999,Z 282.593,A -85,B 0,C 180,E1 -3482.339,E2 -3482.339} C_VEL
LIN {X 0,Y 545.02,Z 282.595,A -85,B 0,C 180,E1 -3484.815,E2 -3484.815} C_VEL
LIN {X 0,Y 545.028,Z 282.595,A -85,B 0,C 180,E1 -3487.241,E2 -3487.241} C_VEL
LIN {X 0,Y 545.1,Z 282.579,A -85,B 0,C 180,E1 -3490.254,E2 -3490.254} C_VEL
LIN {X 0,Y 545.055,Z 282.587,A -85,B 0,C 180,E1 -3492.747,E2 -3492.747} C_VEL
LIN {X 0,Y 545.075,Z 282.584,A -85,B 0,C 180,E1 -3495.818,E2 -3495.818} C_VEL
LIN {X 0,Y 545.115,Z 282.579,A -85,B 0,C 180,E1 -3498.848,E2 -3498.848} C_VEL
LIN {X 0,Y 545.069,Z 282.586,A -85,B 0,C 180,E1 -3501.844,E2 -3501.844} C_VEL
LIN {X 0,Y 545.172,Z 282.571,A -85,B 0,C 180,E1 -3504.821,E2 -3504.821} C_VEL
LIN {X 0,Y 545.192,Z 282.574,A -85,B 0,C 180,E1 -3507.781,E2 -3507.781} C_VEL
LIN {X 0,Y 545.194,Z 282.571,A -85,B 0,C 180,E1 -3509.998,E2 -3509.998} C_VEL
LIN {X 0,Y 545.151,Z 282.573,A -85,B 0,C 180,E1 -3512.953,E2 -3512.953} C_VEL
LIN {X 0,Y 545.134,Z 282.584,A -85,B 0,C 180,E1 -3515.917,E2 -3515.917} C_VEL
LIN {X 0,Y 545.096,Z 282.581,A -85,B 0,C 180,E1 -3518.897,E2 -3518.897} C_VEL
LIN {X 0,Y 545.118,Z 282.587,A -85,B 0,C 180,E1 -3522.279,E2 -3522.279} C_VEL
LIN {X 0,Y 545.127,Z 282.59,A -85,B 0,C 180,E1 -3522.61,E2 -3522.61} C_VEL
LIN {X 0,Y 545.451,Z 289.822,A -85,B 0,C 180,E1 -3523.977,E2 -3523.977} C_VEL
LIN {X 0,Y 545.238,Z 304.214,A -85,B 0,C 180,E1 -3526.663,E2 -3526.663} C_VEL
LIN {X 0,Y 545.19,Z 308.648,A -85,B 0,C 180,E1 -3527.496,E2 -3527.496} C_VEL
LIN {X 0,Y 546.507,Z 316.127,A -85,B 0,C 180,E1 -3527.639,E2 -3527.639} C_VEL
LIN {X 0,Y 546.206,Z 414.751,A -85,B 0,C 180,E1 -3528.955,E2 -3528.955} C_VEL
LIN {X 0,Y 546.07,Z 427.969,A -85,B 0,C 180,E1 -3529.277,E2 -3529.277} C_VEL
LIN {X 0,Y 545.909,Z 440.042,A -85,B 0,C 180,E1 -3529.715,E2 -3529.715} C_VEL
LIN {X 0,Y 545.687,Z 451.764,A -85,B 0,C 180,E1 -3530.285,E2 -3530.285} C_VEL
LIN {X 0,Y 545.477,Z 462.303,A -85,B 0,C 180,E1 -3530.945,E2 -3530.945} C_VEL
LIN {X 0,Y 545.286,Z 473.03,A -85,B 0,C 180,E1 -3531.787,E2 -3531.787} C_VEL
LIN {X 0,Y 545.072,Z 482.964,A -85,B 0,C 180,E1 -3532.752,E2 -3532.752} C_VEL
LIN {X 0,Y 544.921,Z 491.751,A -85,B 0,C 180,E1 -3533.809,E2 -3533.809} C_VEL
LIN {X 0,Y 544.797,Z 499.625,A -85,B 0,C 180,E1 -3534.987,E2 -3534.987} C_VEL
LIN {X 0,Y 544.714,Z 505.163,A -85,B 0,C 180,E1 -3536.015,E2 -3536.015} C_VEL
LIN {X 0,Y 544.642,Z 510.811,A -85,B 0,C 180,E1 -3537.349,E2 -3537.349} C_VEL
LIN {X 0,Y 544.619,Z 514.783,A -85,B 0,C 180,E1 -3538.657,E2 -3538.657} C_VEL
LIN {X 0,Y 544.581,Z 516.357,A -85,B 0,C 180,E1 -3539.362,E2 -3539.362} C_VEL
LIN {X 0,Y 544.58,Z 517.783,A -85,B 0,C 180,E1 -3540.214,E2 -3540.214} C_VEL
LIN {X 0,Y 544.532,Z 518.908,A -85,B 0,C 180,E1 -3541.588,E2 -3541.588} C_VEL
LIN {X 0,Y 544.562,Z 518.66,A -85,B 0,C 180,E1 -3542.978,E2 -3542.978} C_VEL
LIN {X 0,Y 544.571,Z 517.117,A -85,B 0,C 180,E1 -3544.314,E2 -3544.314} C_VEL
LIN {X 0,Y 544.597,Z 514.346,A -85,B 0,C 180,E1 -3545.608,E2 -3545.608} C_VEL
LIN {X 0,Y 544.661,Z 510.326,A -85,B 0,C 180,E1 -3546.868,E2 -3546.868} C_VEL
LIN {X 0,Y 544.719,Z 505.086,A -85,B 0,C 180,E1 -3548.091,E2 -3548.091} C_VEL
LIN {X 0,Y 544.822,Z 498.519,A -85,B 0,C 180,E1 -3549.287,E2 -3549.287} C_VEL
LIN {X 0,Y 544.967,Z 491.587,A -85,B 0,C 180,E1 -3550.303,E2 -3550.303} C_VEL
LIN {X 0,Y 545.108,Z 482.787,A -85,B 0,C 180,E1 -3551.356,E2 -3551.356} C_VEL
LIN {X 0,Y 545.304,Z 472.85,A -85,B 0,C 180,E1 -3552.319,E2 -3552.319} C_VEL
LIN {X 0,Y 545.505,Z 461.752,A -85,B 0,C 180,E1 -3553.184,E2 -3553.184} C_VEL
LIN {X 0,Y 545.75,Z 450.906,A -85,B 0,C 180,E1 -3553.85,E2 -3553.85} C_VEL
LIN {X 0,Y 545.915,Z 438.978,A -85,B 0,C 180,E1 -3554.421,E2 -3554.421} C_VEL
LIN {X 0,Y 546.102,Z 426.2,A -85,B 0,C 180,E1 -3554.868,E2 -3554.868} C_VEL
LIN {X 0,Y 546.205,Z 413.645,A -85,B 0,C 180,E1 -3555.154,E2 -3555.154} C_VEL
LIN {X 0,Y 546.461,Z 316.115,A -85,B 0,C 180,E1 -3556.453,E2 -3556.453} C_VEL
LIN {X 0,Y 545.19,Z 308.482,A -85,B 0,C 180,E1 -3556.605,E2 -3556.605} C_VEL
LIN {X 0,Y 545.284,Z 295.635,A -85,B 0,C 180,E1 -3558.904,E2 -3558.904} C_VEL
LIN {X 0,Y 545.173,Z 283.147,A -85,B 0,C 180,E1 -3561.064,E2 -3561.064} C_VEL
LIN {X 0,Y 545.103,Z 282.585,A -85,B 0,C 180,E1 -3561.176,E2 -3561.176} C_VEL
LIN {X 0,Y 545.024,Z 282.598,A -85,B 0,C 180,E1 -3564.319,E2 -3564.319} C_VEL
LIN {X 0,Y 545.04,Z 282.588,A -85,B 0,C 180,E1 -3567.209,E2 -3567.209} C_VEL
LIN {X 0,Y 545.056,Z 282.588,A -85,B 0,C 180,E1 -3569.81,E2 -3569.81} C_VEL
LIN {X 0,Y 545.055,Z 282.59,A -85,B 0,C 180,E1 -3572.822,E2 -3572.822} C_VEL
LIN {X 0,Y 545.008,Z 282.593,A -85,B 0,C 180,E1 -3575.629,E2 -3575.629} C_VEL
LIN {X 0,Y 545.014,Z 282.596,A -85,B 0,C 180,E1 -3578.834,E2 -3578.834} C_VEL
LIN {X 0,Y 545.03,Z 282.589,A -85,B 0,C 180,E1 -3581.194,E2 -3581.194} C_VEL
LIN {X 0,Y 545.02,Z 282.589,A -85,B 0,C 180,E1 -3583.519,E2 -3583.519} C_VEL
LIN {X 0,Y 545.041,Z 282.587,A -85,B 0,C 180,E1 -3585.818,E2 -3585.818} C_VEL
LIN {X 0,Y 545.079,Z 282.588,A -85,B 0,C 180,E1 -3588.848,E2 -3588.848} C_VEL
LIN {X 0,Y 545.075,Z 282.582,A -85,B 0,C 180,E1 -3591.846,E2 -3591.846} C_VEL
LIN {X 0,Y 545.154,Z 282.581,A -85,B 0,C 180,E1 -3594.822,E2 -3594.822} C_VEL
LIN {X 0,Y 545.134,Z 282.575,A -85,B 0,C 180,E1 -3597.783,E2 -3597.783} C_VEL
LIN {X 0,Y 545.168,Z 282.576,A -85,B 0,C 180,E1 -3600.739,E2 -3600.739} C_VEL
LIN {X 0,Y 545.13,Z 282.583,A -85,B 0,C 180,E1 -3602.956,E2 -3602.956} C_VEL
LIN {X 0,Y 545.123,Z 282.576,A -85,B 0,C 180,E1 -3605.92,E2 -3605.92} C_VEL
LIN {X 0,Y 545.081,Z 282.588,A -85,B 0,C 180,E1 -3608.901,E2 -3608.901} C_VEL
LIN {X 0,Y 545.084,Z 282.579,A -85,B 0,C 180,E1 -3611.905,E2 -3611.905} C_VEL
LIN {X 0,Y 545.055,Z 282.591,A -85,B 0,C 180,E1 -3614.944,E2 -3614.944} C_VEL
LIN {X 0,Y 545.048,Z 282.585,A -85,B 0,C 180,E1 -3618.027,E2 -3618.027} C_VEL
LIN {X 0,Y 545.052,Z 282.583,A -85,B 0,C 180,E1 -3620.374,E2 -3620.374} C_VEL
LIN {X 0,Y 545.097,Z 282.583,A -85,B 0,C 180,E1 -3623.559,E2 -3623.559} C_VEL
LIN {X 0,Y 545.067,Z 282.584,A -85,B 0,C 180,E1 -3626.001,E2 -3626.001} C_VEL
LIN {X 0,Y 545.06,Z 282.583,A -85,B 0,C 180,E1 -3628.755,E2 -3628.755} C_VEL
LIN {X 0,Y 545.037,Z 282.593,A -85,B 0,C 180,E1 -3631.686,E2 -3631.686} C_VEL
LIN {X 0,Y 545.047,Z 282.585,A -85,B 0,C 180,E1 -3634.566,E2 -3634.566} C_VEL
LIN {X 0,Y 545.053,Z 282.591,A -85,B 0,C 180,E1 -3637.303,E2 -3637.303} C_VEL
LIN {X 0,Y 545.114,Z 282.58,A -85,B 0,C 180,E1 -3640.139,E2 -3640.139} C_VEL
LIN {X 0,Y 545.056,Z 282.588,A -85,B 0,C 180,E1 -3643.109,E2 -3643.109} C_VEL
LIN {X 0,Y 545.036,Z 282.591,A -85,B 0,C 180,E1 -3646.228,E2 -3646.228} C_VEL
LIN {X 0,Y 545.096,Z 282.581,A -85,B 0,C 180,E1 -3648.893,E2 -3648.893} C_VEL
LIN {X 0,Y 545.033,Z 282.598,A -85,B 0,C 180,E1 -3651.767,E2 -3651.767} C_VEL
LIN {X 0,Y 545.044,Z 282.589,A -85,B 0,C 180,E1 -3654.538,E2 -3654.538} C_VEL
LIN {X 0,Y 545.063,Z 282.587,A -85,B 0,C 180,E1 -3657.217,E2 -3657.217} C_VEL
LIN {X 0,Y 545.084,Z 282.591,A -85,B 0,C 180,E1 -3659.817,E2 -3659.817} C_VEL
LIN {X 0,Y 545.088,Z 282.583,A -85,B 0,C 180,E1 -3662.828,E2 -3662.828} C_VEL
LIN {X 0,Y 545.069,Z 282.59,A -85,B 0,C 180,E1 -3665.636,E2 -3665.636} C_VEL
LIN {X 0,Y 545.127,Z 282.661,A -85,B 0,C 180,E1 -3666.014,E2 -3666.014} C_VEL
LIN {X 0,Y 546.233,Z 289.628,A -85,B 0,C 180,E1 -3667.099,E2 -3667.099} C_VEL
LIN {X 0,Y 545.846,Z 312.165,A -85,B 0,C 180,E1 -3670.446,E2 -3670.446} C_VEL
LIN {X 0,Y 545.533,Z 330.661,A -85,B 0,C 180,E1 -3673.154,E2 -3673.154} C_VEL
LIN {X 0,Y 545.35,Z 346.394,A -85,B 0,C 180,E1 -3675.437,E2 -3675.437} C_VEL
LIN {X 0,Y 546.529,Z 355.508,A -85,B 0,C 180,E1 -3675.593,E2 -3675.593} C_VEL
LIN {X 0,Y 546.19,Z 454.92,A -85,B 0,C 180,E1 -3676.919,E2 -3676.919} C_VEL
LIN {X 0,Y 546.024,Z 468.184,A -85,B 0,C 180,E1 -3677.246,E2 -3677.246} C_VEL
LIN {X 0,Y 545.871,Z 480.354,A -85,B 0,C 180,E1 -3677.691,E2 -3677.691} C_VEL
LIN {X 0,Y 545.759,Z 491.266,A -85,B 0,C 180,E1 -3678.224,E2 -3678.224} C_VEL
LIN {X 0,Y 545.529,Z 502.945,A -85,B 0,C 180,E1 -3678.955,E2 -3678.955} C_VEL
LIN {X 0,Y 545.277,Z 513.571,A -85,B 0,C 180,E1 -3679.795,E2 -3679.795} C_VEL
LIN {X 0,Y 545.082,Z 523.143,A -85,B 0,C 180,E1 -3680.728,E2 -3680.728} C_VEL
LIN {X 0,Y 544.976,Z 530.984,A -85,B 0,C 180,E1 -3681.661,E2 -3681.661} C_VEL
LIN {X 0,Y 544.821,Z 538.639,A -85,B 0,C 180,E1 -3682.778,E2 -3682.778} C_VEL
LIN {X 0,Y 544.78,Z 545.693,A -85,B 0,C 180,E1 -3684.079,E2 -3684.079} C_VEL
LIN {X 0,Y 544.628,Z 550.383,A -85,B 0,C 180,E1 -3685.191,E2 -3685.191} C_VEL
LIN {X 0,Y 544.668,Z 553.966,A -85,B 0,C 180,E1 -3686.304,E2 -3686.304} C_VEL
LIN {X 0,Y 544.65,Z 555.812,A -85,B 0,C 180,E1 -3687.044,E2 -3687.044} C_VEL
LIN {X 0,Y 544.545,Z 558.185,A -85,B 0,C 180,E1 -3688.523,E2 -3688.523} C_VEL
LIN {X 0,Y 544.541,Z 559,A -85,B 0,C 180,E1 -3690.002,E2 -3690.002} C_VEL
LIN {X 0,Y 544.546,Z 558.181,A -85,B 0,C 180,E1 -3691.481,E2 -3691.481} C_VEL
LIN {X 0,Y 544.651,Z 555.805,A -85,B 0,C 180,E1 -3692.961,E2 -3692.961} C_VEL
LIN {X 0,Y 544.684,Z 552.889,A -85,B 0,C 180,E1 -3694.072,E2 -3694.072} C_VEL
LIN {X 0,Y 544.654,Z 548.94,A -85,B 0,C 180,E1 -3695.184,E2 -3695.184} C_VEL
LIN {X 0,Y 544.74,Z 543.585,A -85,B 0,C 180,E1 -3696.351,E2 -3696.351} C_VEL
LIN {X 0,Y 544.861,Z 536.223,A -85,B 0,C 180,E1 -3697.599,E2 -3697.599} C_VEL
LIN {X 0,Y 545.018,Z 527.977,A -85,B 0,C 180,E1 -3698.717,E2 -3698.717} C_VEL
LIN {X 0,Y 545.203,Z 519.522,A -85,B 0,C 180,E1 -3699.649,E2 -3699.649} C_VEL
LIN {X 0,Y 545.371,Z 509.069,A -85,B 0,C 180,E1 -3700.583,E2 -3700.583} C_VEL
LIN {X 0,Y 545.613,Z 497.465,A -85,B 0,C 180,E1 -3701.412,E2 -3701.412} C_VEL
LIN {X 0,Y 545.798,Z 487.315,A -85,B 0,C 180,E1 -3701.985,E2 -3701.985} C_VEL
LIN {X 0,Y 545.943,Z 475.615,A -85,B 0,C 180,E1 -3702.501,E2 -3702.501} C_VEL
LIN {X 0,Y 546.106,Z 462.133,A -85,B 0,C 180,E1 -3702.922,E2 -3702.922} C_VEL
LIN {X 0,Y 546.249,Z 448.767,A -85,B 0,C 180,E1 -3703.179,E2 -3703.179} C_VEL
LIN {X 0,Y 546.463,Z 353.71,A -85,B 0,C 180,E1 -3704.433,E2 -3704.433} C_VEL
LIN {X 0,Y 545.362,Z 346.459,A -85,B 0,C 180,E1 -3704.567,E2 -3704.567} C_VEL
LIN {X 0,Y 545.715,Z 322.964,A -85,B 0,C 180,E1 -3708.005,E2 -3708.005} C_VEL
LIN {X 0,Y 545.983,Z 304.584,A -85,B 0,C 180,E1 -3710.732,E2 -3710.732} C_VEL
LIN {X 0,Y 546.241,Z 288.845,A -85,B 0,C 180,E1 -3713.106,E2 -3713.106} C_VEL
LIN {X 0,Y 545.093,Z 282.587,A -85,B 0,C 180,E1 -3714.123,E2 -3714.123} C_VEL
LIN {X 0,Y 545.085,Z 282.584,A -85,B 0,C 180,E1 -3717.171,E2 -3717.171} C_VEL
LIN {X 0,Y 545.082,Z 282.589,A -85,B 0,C 180,E1 -3720.247,E2 -3720.247} C_VEL
LIN {X 0,Y 545.082,Z 282.581,A -85,B 0,C 180,E1 -3723.062,E2 -3723.062} C_VEL
LIN {X 0,Y 545.035,Z 282.589,A -85,B 0,C 180,E1 -3725.673,E2 -3725.673} C_VEL
LIN {X 0,Y 545.053,Z 282.595,A -85,B 0,C 180,E1 -3728.237,E2 -3728.237} C_VEL
LIN {X 0,Y 545.086,Z 282.581,A -85,B 0,C 180,E1 -3731.114,E2 -3731.114} C_VEL
LIN {X 0,Y 545.048,Z 282.591,A -85,B 0,C 180,E1 -3734.13,E2 -3734.13} C_VEL
LIN {X 0,Y 545.061,Z 282.584,A -85,B 0,C 180,E1 -3737.303,E2 -3737.303} C_VEL
LIN {X 0,Y 545.068,Z 282.584,A -85,B 0,C 180,E1 -3739.857,E2 -3739.857} C_VEL
LIN {X 0,Y 545.069,Z 282.586,A -85,B 0,C 180,E1 -3743.073,E2 -3743.073} C_VEL
LIN {X 0,Y 545.063,Z 282.588,A -85,B 0,C 180,E1 -3746.328,E2 -3746.328} C_VEL
LIN {X 0,Y 545.064,Z 282.59,A -85,B 0,C 180,E1 -3748.952,E2 -3748.952} C_VEL
LIN {X 0,Y 545.094,Z 282.58,A -85,B 0,C 180,E1 -3751.507,E2 -3751.507} C_VEL
LIN {X 0,Y 545.091,Z 282.584,A -85,B 0,C 180,E1 -3754.49,E2 -3754.49} C_VEL
LIN {X 0,Y 545.034,Z 282.592,A -85,B 0,C 180,E1 -3757.242,E2 -3757.242} C_VEL
LIN {X 0,Y 545.109,Z 282.579,A -85,B 0,C 180,E1 -3760.414,E2 -3760.414} C_VEL
LIN {X 0,Y 545.06,Z 282.587,A -85,B 0,C 180,E1 -3763.521,E2 -3763.521} C_VEL
LIN {X 0,Y 545.083,Z 282.582,A -85,B 0,C 180,E1 -3765.82,E2 -3765.82} C_VEL
LIN {X 0,Y 545.11,Z 282.582,A -85,B 0,C 180,E1 -3768.849,E2 -3768.849} C_VEL
LIN {X 0,Y 545.114,Z 282.579,A -85,B 0,C 180,E1 -3771.847,E2 -3771.847} C_VEL
LIN {X 0,Y 545.195,Z 282.569,A -85,B 0,C 180,E1 -3774.823,E2 -3774.823} C_VEL
LIN {X 0,Y 545.176,Z 282.574,A -85,B 0,C 180,E1 -3777.784,E2 -3777.784} C_VEL
LIN {X 0,Y 545.197,Z 282.567,A -85,B 0,C 180,E1 -3780.739,E2 -3780.739} C_VEL
LIN {X 0,Y 545.157,Z 282.573,A -85,B 0,C 180,E1 -3782.956,E2 -3782.956} C_VEL
LIN {X 0,Y 545.147,Z 282.578,A -85,B 0,C 180,E1 -3785.92,E2 -3785.92} C_VEL
LIN {X 0,Y 545.093,Z 282.58,A -85,B 0,C 180,E1 -3788.901,E2 -3788.901} C_VEL
LIN {X 0,Y 545.091,Z 282.588,A -85,B 0,C 180,E1 -3791.905,E2 -3791.905} C_VEL
LIN {X 0,Y 545.068,Z 282.583,A -85,B 0,C 180,E1 -3794.944,E2 -3794.944} C_VEL
LIN {X 0,Y 545.05,Z 282.593,A -85,B 0,C 180,E1 -3798.027,E2 -3798.027} C_VEL
LIN {X 0,Y 545.078,Z 282.585,A -85,B 0,C 180,E1 -3800.373,E2 -3800.373} C_VEL
LIN {X 0,Y 545.064,Z 282.586,A -85,B 0,C 180,E1 -3803.56,E2 -3803.56} C_VEL
LIN {X 0,Y 545.031,Z 282.596,A -85,B 0,C 180,E1 -3806.003,E2 -3806.003} C_VEL
LIN {X 0,Y 545.013,Z 282.592,A -85,B 0,C 180,E1 -3808.736,E2 -3808.736} C_VEL
LIN {X 0,Y 545.054,Z 282.585,A -85,B 0,C 180,E1 -3811.049,E2 -3811.049} C_VEL
LIN {X 0,Y 545.035,Z 282.589,A -85,B 0,C 180,E1 -3813.767,E2 -3813.767} C_VEL
LIN {X 0,Y 544.996,Z 282.602,A -85,B 0,C 180,E1 -3816.384,E2 -3816.384} C_VEL
LIN {X 0,Y 544.994,Z 282.593,A -85,B 0,C 180,E1 -3816.984,E2 -3816.984} C_VEL
LIN {X 0,Y 544.333,Z 282.675,A -85,B 0,C 180,E1 -3817.601,E2 -3817.601} C_VEL
LIN {X 0,Y 541.474,Z 283.037,A -85,B 0,C 180,E1 -3818.602,E2 -3818.602} C_VEL
LIN {X 0,Y 539.061,Z 283.334,A -85,B 0,C 180,E1 -3819.408,E2 -3819.408} C_VEL
LIN {X 0,Y 538.035,Z 283.463,A -85,B 0,C 180,E1 -3820.031,E2 -3820.031} C_VEL
LIN {X 0,Y 537.957,Z 283.47,A -85,B 0,C 180,E1 -3820.241,E2 -3820.241} C_VEL
LIN {X 0,Y 537.95,Z 283.472,A -85,B 0,C 180,E1 -3822.979,E2 -3822.979} C_VEL
LIN {X 0,Y 537.993,Z 283.465,A -85,B 0,C 180,E1 -3825.93,E2 -3825.93} C_VEL
LIN {X 0,Y 537.975,Z 283.47,A -85,B 0,C 180,E1 -3828.222,E2 -3828.222} C_VEL
LIN {X 0,Y 537.966,Z 283.471,A -85,B 0,C 180,E1 -3831.166,E2 -3831.166} C_VEL
LIN {X 0,Y 537.937,Z 283.472,A -85,B 0,C 180,E1 -3834.098,E2 -3834.098} C_VEL
LIN {X 0,Y 537.984,Z 283.474,A -85,B 0,C 180,E1 -3836.728,E2 -3836.728} C_VEL
LIN {X 0,Y 537.99,Z 283.466,A -85,B 0,C 180,E1 -3839.563,E2 -3839.563} C_VEL
LIN {X 0,Y 537.991,Z 283.469,A -85,B 0,C 180,E1 -3842.662,E2 -3842.662} C_VEL
LIN {X 0,Y 537.968,Z 283.473,A -85,B 0,C 180,E1 -3845.288,E2 -3845.288} C_VEL
LIN {X 0,Y 538.019,Z 283.461,A -85,B 0,C 180,E1 -3848.042,E2 -3848.042} C_VEL
LIN {X 0,Y 537.997,Z 283.47,A -85,B 0,C 180,E1 -3850.937,E2 -3850.937} C_VEL
LIN {X 0,Y 537.991,Z 283.474,A -85,B 0,C 180,E1 -3853.297,E2 -3853.297} C_VEL
LIN {X 0,Y 538.048,Z 283.462,A -85,B 0,C 180,E1 -3855.629,E2 -3855.629} C_VEL
LIN {X 0,Y 538.077,Z 283.455,A -85,B 0,C 180,E1 -3858.7,E2 -3858.7} C_VEL
LIN {X 0,Y 538.038,Z 283.464,A -85,B 0,C 180,E1 -3861.737,E2 -3861.737} C_VEL
LIN {X 0,Y 538.13,Z 283.448,A -85,B 0,C 180,E1 -3864.753,E2 -3864.753} C_VEL
LIN {X 0,Y 538.164,Z 283.45,A -85,B 0,C 180,E1 -3867.752,E2 -3867.752} C_VEL
LIN {X 0,Y 538.162,Z 283.447,A -85,B 0,C 180,E1 -3869.998,E2 -3869.998} C_VEL
LIN {X 0,Y 538.118,Z 283.449,A -85,B 0,C 180,E1 -3872.992,E2 -3872.992} C_VEL
LIN {X 0,Y 538.09,Z 283.46,A -85,B 0,C 180,E1 -3875.995,E2 -3875.995} C_VEL
LIN {X 0,Y 538.048,Z 283.459,A -85,B 0,C 180,E1 -3879.015,E2 -3879.015} C_VEL
LIN {X 0,Y 538.071,Z 283.465,A -85,B 0,C 180,E1 -3882.059,E2 -3882.059} C_VEL
LIN {X 0,Y 538.112,Z 283.587,A -85,B 0,C 180,E1 -3882.537,E2 -3882.537} C_VEL
LIN {X 0,Y 538.444,Z 290.094,A -85,B 0,C 180,E1 -3883.777,E2 -3883.777} C_VEL
LIN {X 0,Y 538.254,Z 304.558,A -85,B 0,C 180,E1 -3886.495,E2 -3886.495} C_VEL
LIN {X 0,Y 538.205,Z 308.856,A -85,B 0,C 180,E1 -3887.303,E2 -3887.303} C_VEL
LIN {X 0,Y 539.683,Z 317.884,A -85,B 0,C 180,E1 -3887.474,E2 -3887.474} C_VEL
LIN {X 0,Y 539.28,Z 415.714,A -85,B 0,C 180,E1 -3888.801,E2 -3888.801} C_VEL
LIN {X 0,Y 539.156,Z 429.031,A -85,B 0,C 180,E1 -3889.138,E2 -3889.138} C_VEL
LIN {X 0,Y 538.955,Z 441.724,A -85,B 0,C 180,E1 -3889.616,E2 -3889.616} C_VEL
LIN {X 0,Y 538.727,Z 453.05,A -85,B 0,C 180,E1 -3890.194,E2 -3890.194} C_VEL
LIN {X 0,Y 538.479,Z 464.291,A -85,B 0,C 180,E1 -3890.93,E2 -3890.93} C_VEL
LIN {X 0,Y 538.288,Z 474.481,A -85,B 0,C 180,E1 -3891.762,E2 -3891.762} C_VEL
LIN {X 0,Y 538.058,Z 483.477,A -85,B 0,C 180,E1 -3892.659,E2 -3892.659} C_VEL
LIN {X 0,Y 537.902,Z 491.708,A -85,B 0,C 180,E1 -3893.663,E2 -3893.663} C_VEL
LIN {X 0,Y 537.779,Z 498.756,A -85,B 0,C 180,E1 -3894.716,E2 -3894.716} C_VEL
LIN {X 0,Y 537.646,Z 505.453,A -85,B 0,C 180,E1 -3895.965,E2 -3895.965} C_VEL
LIN {X 0,Y 537.576,Z 510.791,A -85,B 0,C 180,E1 -3897.252,E2 -3897.252} C_VEL
LIN {X 0,Y 537.52,Z 513.422,A -85,B 0,C 180,E1 -3898.075,E2 -3898.075} C_VEL
LIN {X 0,Y 537.498,Z 515.611,A -85,B 0,C 180,E1 -3898.928,E2 -3898.928} C_VEL
LIN {X 0,Y 537.49,Z 518.026,A -85,B 0,C 180,E1 -3900.346,E2 -3900.346} C_VEL
LIN {X 0,Y 537.442,Z 519.003,A -85,B 0,C 180,E1 -3901.789,E2 -3901.789} C_VEL
LIN {X 0,Y 537.448,Z 518.489,A -85,B 0,C 180,E1 -3903.308,E2 -3903.308} C_VEL
LIN {X 0,Y 537.468,Z 516.867,A -85,B 0,C 180,E1 -3904.533,E2 -3904.533} C_VEL
LIN {X 0,Y 537.528,Z 513.91,A -85,B 0,C 180,E1 -3905.842,E2 -3905.842} C_VEL
LIN {X 0,Y 537.585,Z 509.772,A -85,B 0,C 180,E1 -3907.11,E2 -3907.11} C_VEL
LIN {X 0,Y 537.672,Z 504.402,A -85,B 0,C 180,E1 -3908.346,E2 -3908.346} C_VEL
LIN {X 0,Y 537.821,Z 497.641,A -85,B 0,C 180,E1 -3909.557,E2 -3909.557} C_VEL
LIN {X 0,Y 537.962,Z 489.327,A -85,B 0,C 180,E1 -3910.736,E2 -3910.736} C_VEL
LIN {X 0,Y 538.137,Z 480.435,A -85,B 0,C 180,E1 -3911.756,E2 -3911.756} C_VEL
LIN {X 0,Y 538.337,Z 471.086,A -85,B 0,C 180,E1 -3912.63,E2 -3912.63} C_VEL
LIN {X 0,Y 538.581,Z 460.216,A -85,B 0,C 180,E1 -3913.448,E2 -3913.448} C_VEL
LIN {X 0,Y 538.864,Z 448.132,A -85,B 0,C 180,E1 -3914.166,E2 -3914.166} C_VEL
LIN {X 0,Y 539.049,Z 436.259,A -85,B 0,C 180,E1 -3914.702,E2 -3914.702} C_VEL
LIN {X 0,Y 539.2,Z 423.616,A -85,B 0,C 180,E1 -3915.109,E2 -3915.109} C_VEL
LIN {X 0,Y 539.353,Z 410.906,A -85,B 0,C 180,E1 -3915.369,E2 -3915.369} C_VEL
LIN {X 0,Y 539.564,Z 316.796,A -85,B 0,C 180,E1 -3916.634,E2 -3916.634} C_VEL
LIN {X 0,Y 538.178,Z 308.655,A -85,B 0,C 180,E1 -3916.786,E2 -3916.786} C_VEL
LIN {X 0,Y 538.241,Z 294.853,A -85,B 0,C 180,E1 -3919.242,E2 -3919.242} C_VEL
LIN {X 0,Y 538.207,Z 284.97,A -85,B 0,C 180,E1 -3920.945,E2 -3920.945} C_VEL
LIN {X 0,Y 538.064,Z 283.462,A -85,B 0,C 180,E1 -3921.242,E2 -3921.242} C_VEL
LIN {X 0,Y 537.99,Z 283.474,A -85,B 0,C 180,E1 -3924.08,E2 -3924.08} C_VEL
LIN {X 0,Y 537.994,Z 283.469,A -85,B 0,C 180,E1 -3926.725,E2 -3926.725} C_VEL
LIN {X 0,Y 537.993,Z 283.466,A -85,B 0,C 180,E1 -3929.551,E2 -3929.551} C_VEL
LIN {X 0,Y 538.002,Z 283.468,A -85,B 0,C 180,E1 -3931.948,E2 -3931.948} C_VEL
LIN {X 0,Y 538.044,Z 283.469,A -85,B 0,C 180,E1 -3934.466,E2 -3934.466} C_VEL
LIN {X 0,Y 537.945,Z 283.473,A -85,B 0,C 180,E1 -3937.736,E2 -3937.736} C_VEL
LIN {X 0,Y 538.027,Z 283.466,A -85,B 0,C 180,E1 -3940.146,E2 -3940.146} C_VEL
LIN {X 0,Y 537.971,Z 283.468,A -85,B 0,C 180,E1 -3943.297,E2 -3943.297} C_VEL
LIN {X 0,Y 538.009,Z 283.463,A -85,B 0,C 180,E1 -3945.629,E2 -3945.629} C_VEL
LIN {X 0,Y 538.035,Z 283.467,A -85,B 0,C 180,E1 -3948.701,E2 -3948.701} C_VEL
LIN {X 0,Y 538.032,Z 283.46,A -85,B 0,C 180,E1 -3951.739,E2 -3951.739} C_VEL
LIN {X 0,Y 538.13,Z 283.457,A -85,B 0,C 180,E1 -3954.755,E2 -3954.755} C_VEL
LIN {X 0,Y 538.106,Z 283.45,A -85,B 0,C 180,E1 -3957.754,E2 -3957.754} C_VEL
LIN {X 0,Y 538.137,Z 283.452,A -85,B 0,C 180,E1 -3960.748,E2 -3960.748} C_VEL
LIN {X 0,Y 538.095,Z 283.458,A -85,B 0,C 180,E1 -3962.995,E2 -3962.995} C_VEL
LIN {X 0,Y 538.074,Z 283.454,A -85,B 0,C 180,E1 -3965.998,E2 -3965.998} C_VEL
LIN {X 0,Y 538.031,Z 283.468,A -85,B 0,C 180,E1 -3969.018,E2 -3969.018} C_VEL
LIN {X 0,Y 538.032,Z 283.457,A -85,B 0,C 180,E1 -3972.064,E2 -3972.064} C_VEL
LIN {X 0,Y 538.006,Z 283.471,A -85,B 0,C 180,E1 -3975.145,E2 -3975.145} C_VEL
LIN {X 0,Y 537.997,Z 283.463,A -85,B 0,C 180,E1 -3978.271,E2 -3978.271} C_VEL
LIN {X 0,Y 537.997,Z 283.463,A -85,B 0,C 180,E1 -3980.653,E2 -3980.653} C_VEL
LIN {X 0,Y 538.025,Z 283.466,A -85,B 0,C 180,E1 -3983.071,E2 -3983.071} C_VEL
LIN {X 0,Y 538.03,Z 283.464,A -85,B 0,C 180,E1 -3985.683,E2 -3985.683} C_VEL
LIN {X 0,Y 538.013,Z 283.461,A -85,B 0,C 180,E1 -3988.052,E2 -3988.052} C_VEL
LIN {X 0,Y 537.984,Z 283.466,A -85,B 0,C 180,E1 -3990.629,E2 -3990.629} C_VEL
LIN {X 0,Y 538.002,Z 283.469,A -85,B 0,C 180,E1 -3993.286,E2 -3993.286} C_VEL
LIN {X 0,Y 537.998,Z 283.467,A -85,B 0,C 180,E1 -3996.004,E2 -3996.004} C_VEL
LIN {X 0,Y 537.998,Z 283.464,A -85,B 0,C 180,E1 -3998.832,E2 -3998.832} C_VEL
LIN {X 0,Y 538.049,Z 283.458,A -85,B 0,C 180,E1 -4000.776,E2 -4000.776} C_VEL
LIN {X 0,Y 537.997,Z 283.47,A -85,B 0,C 180,E1 -4004.079,E2 -4004.079} C_VEL
LIN {X 0,Y 537.996,Z 283.468,A -85,B 0,C 180,E1 -4007.219,E2 -4007.219} C_VEL
LIN {X 0,Y 538.03,Z 283.465,A -85,B 0,C 180,E1 -4010.21,E2 -4010.21} C_VEL
LIN {X 0,Y 538.011,Z 283.463,A -85,B 0,C 180,E1 -4013.072,E2 -4013.072} C_VEL
LIN {X 0,Y 538.013,Z 283.473,A -85,B 0,C 180,E1 -4015.832,E2 -4015.832} C_VEL
LIN {X 0,Y 538.006,Z 283.468,A -85,B 0,C 180,E1 -4018.504,E2 -4018.504} C_VEL
LIN {X 0,Y 538.043,Z 283.461,A -85,B 0,C 180,E1 -4021.104,E2 -4021.104} C_VEL
LIN {X 0,Y 538.037,Z 283.465,A -85,B 0,C 180,E1 -4023.638,E2 -4023.638} C_VEL
LIN {X 0,Y 538.068,Z 283.578,A -85,B 0,C 180,E1 -4025.879,E2 -4025.879} C_VEL
LIN {X 0,Y 539.27,Z 290.585,A -85,B 0,C 180,E1 -4026.989,E2 -4026.989} C_VEL
LIN {X 0,Y 538.907,Z 311.849,A -85,B 0,C 180,E1 -4030.184,E2 -4030.184} C_VEL
LIN {X 0,Y 538.513,Z 331.666,A -85,B 0,C 180,E1 -4033.123,E2 -4033.123} C_VEL
LIN {X 0,Y 538.316,Z 346.089,A -85,B 0,C 180,E1 -4035.241,E2 -4035.241} C_VEL
LIN {X 0,Y 539.678,Z 356.443,A -85,B 0,C 180,E1 -4035.424,E2 -4035.424} C_VEL
LIN {X 0,Y 539.276,Z 454.518,A -85,B 0,C 180,E1 -4036.748,E2 -4036.748} C_VEL
LIN {X 0,Y 539.096,Z 467.821,A -85,B 0,C 180,E1 -4037.079,E2 -4037.079} C_VEL
LIN {X 0,Y 538.872,Z 480.01,A -85,B 0,C 180,E1 -4037.529,E2 -4037.529} C_VEL
LIN {X 0,Y 538.777,Z 491.523,A -85,B 0,C 180,E1 -4038.101,E2 -4038.101} C_VEL
LIN {X 0,Y 538.541,Z 502.643,A -85,B 0,C 180,E1 -4038.81,E2 -4038.81} C_VEL
LIN {X 0,Y 538.251,Z 513.33,A -85,B 0,C 180,E1 -4039.661,E2 -4039.661} C_VEL
LIN {X 0,Y 538.065,Z 522.964,A -85,B 0,C 180,E1 -4040.606,E2 -4040.606} C_VEL
LIN {X 0,Y 537.921,Z 530.861,A -85,B 0,C 180,E1 -4041.551,E2 -4041.551} C_VEL
LIN {X 0,Y 537.752,Z 538.571,A -85,B 0,C 180,E1 -4042.682,E2 -4042.682} C_VEL
LIN {X 0,Y 537.697,Z 545.681,A -85,B 0,C 180,E1 -4044.001,E2 -4044.001} C_VEL
LIN {X 0,Y 537.54,Z 550.383,A -85,B 0,C 180,E1 -4045.128,E2 -4045.128} C_VEL
LIN {X 0,Y 537.59,Z 553.965,A -85,B 0,C 180,E1 -4046.255,E2 -4046.255} C_VEL
LIN {X 0,Y 537.55,Z 555.812,A -85,B 0,C 180,E1 -4047.005,E2 -4047.005} C_VEL
LIN {X 0,Y 537.451,Z 558.184,A -85,B 0,C 180,E1 -4048.504,E2 -4048.504} C_VEL
LIN {X 0,Y 537.442,Z 559,A -85,B 0,C 180,E1 -4050.002,E2 -4050.002} C_VEL
LIN {X 0,Y 537.451,Z 558.181,A -85,B 0,C 180,E1 -4051.501,E2 -4051.501} C_VEL
LIN {X 0,Y 537.551,Z 555.805,A -85,B 0,C 180,E1 -4053,E2 -4053} C_VEL
LIN {X 0,Y 537.604,Z 552.889,A -85,B 0,C 180,E1 -4054.125,E2 -4054.125} C_VEL
LIN {X 0,Y 537.588,Z 548.939,A -85,B 0,C 180,E1 -4055.253,E2 -4055.253} C_VEL
LIN {X 0,Y 537.653,Z 544.049,A -85,B 0,C 180,E1 -4056.336,E2 -4056.336} C_VEL
LIN {X 0,Y 537.774,Z 537.379,A -85,B 0,C 180,E1 -4057.511,E2 -4057.511} C_VEL
LIN {X 0,Y 537.943,Z 529.335,A -85,B 0,C 180,E1 -4058.643,E2 -4058.643} C_VEL
LIN {X 0,Y 538.116,Z 521.137,A -85,B 0,C 180,E1 -4059.587,E2 -4059.587} C_VEL
LIN {X 0,Y 538.335,Z 511.14,A -85,B 0,C 180,E1 -4060.533,E2 -4060.533} C_VEL
LIN {X 0,Y 538.595,Z 501.278,A -85,B 0,C 180,E1 -4061.289,E2 -4061.289} C_VEL
LIN {X 0,Y 538.732,Z 490.164,A -85,B 0,C 180,E1 -4061.975,E2 -4061.975} C_VEL
LIN {X 0,Y 538.952,Z 477.652,A -85,B 0,C 180,E1 -4062.57,E2 -4062.57} C_VEL
LIN {X 0,Y 539.153,Z 464.533,A -85,B 0,C 180,E1 -4063.02,E2 -4063.02} C_VEL
LIN {X 0,Y 539.303,Z 451.405,A -85,B 0,C 180,E1 -4063.304,E2 -4063.304} C_VEL
LIN {X 0,Y 539.529,Z 354.006,A -85,B 0,C 180,E1 -4064.614,E2 -4064.614} C_VEL
LIN {X 0,Y 538.342,Z 346.199,A -85,B 0,C 180,E1 -4064.763,E2 -4064.763} C_VEL
LIN {X 0,Y 538.722,Z 323.804,A -85,B 0,C 180,E1 -4068.087,E2 -4068.087} C_VEL
LIN {X 0,Y 539.018,Z 305.668,A -85,B 0,C 180,E1 -4070.813,E2 -4070.813} C_VEL
LIN {X 0,Y 539.355,Z 291.26,A -85,B 0,C 180,E1 -4073.012,E2 -4073.012} C_VEL
LIN {X 0,Y 538.051,Z 283.464,A -85,B 0,C 180,E1 -4074.297,E2 -4074.297} C_VEL
LIN {X 0,Y 538.055,Z 283.46,A -85,B 0,C 180,E1 -4077.205,E2 -4077.205} C_VEL
LIN {X 0,Y 538.019,Z 283.468,A -85,B 0,C 180,E1 -4079.762,E2 -4079.762} C_VEL
LIN {X 0,Y 538.022,Z 283.466,A -85,B 0,C 180,E1 -4082.383,E2 -4082.383} C_VEL
LIN {X 0,Y 538,Z 283.463,A -85,B 0,C 180,E1 -4085.084,E2 -4085.084} C_VEL
LIN {X 0,Y 537.993,Z 283.468,A -85,B 0,C 180,E1 -4087.878,E2 -4087.878} C_VEL
LIN {X 0,Y 538.049,Z 283.46,A -85,B 0,C 180,E1 -4090.775,E2 -4090.775} C_VEL
LIN {X 0,Y 538.002,Z 283.465,A -85,B 0,C 180,E1 -4093.816,E2 -4093.816} C_VEL
LIN {X 0,Y 538.024,Z 283.462,A -85,B 0,C 180,E1 -4097.012,E2 -4097.012} C_VEL
LIN {X 0,Y 538.049,Z 283.458,A -85,B 0,C 180,E1 -4099.252,E2 -4099.252} C_VEL
LIN {X 0,Y 537.989,Z 283.468,A -85,B 0,C 180,E1 -4102.122,E2 -4102.122} C_VEL
LIN {X 0,Y 538.006,Z 283.468,A -85,B 0,C 180,E1 -4104.916,E2 -4104.916} C_VEL
LIN {X 0,Y 538.025,Z 283.46,A -85,B 0,C 180,E1 -4107.618,E2 -4107.618} C_VEL
LIN {X 0,Y 538.036,Z 283.461,A -85,B 0,C 180,E1 -4110.24,E2 -4110.24} C_VEL
LIN {X 0,Y 538.06,Z 283.465,A -85,B 0,C 180,E1 -4112.796,E2 -4112.796} C_VEL
LIN {X 0,Y 538.04,Z 283.462,A -85,B 0,C 180,E1 -4115.292,E2 -4115.292} C_VEL
LIN {X 0,Y 538.006,Z 283.462,A -85,B 0,C 180,E1 -4118.042,E2 -4118.042} C_VEL
LIN {X 0,Y 538.026,Z 283.469,A -85,B 0,C 180,E1 -4120.94,E2 -4120.94} C_VEL
LIN {X 0,Y 538.012,Z 283.468,A -85,B 0,C 180,E1 -4123.299,E2 -4123.299} C_VEL
LIN {X 0,Y 538.052,Z 283.46,A -85,B 0,C 180,E1 -4125.63,E2 -4125.63} C_VEL
LIN {X 0,Y 538.068,Z 283.457,A -85,B 0,C 180,E1 -4128.701,E2 -4128.701} C_VEL
LIN {X 0,Y 538.071,Z 283.457,A -85,B 0,C 180,E1 -4131.739,E2 -4131.739} C_VEL
LIN {X 0,Y 538.152,Z 283.446,A -85,B 0,C 180,E1 -4134.755,E2 -4134.755} C_VEL
LIN {X 0,Y 538.149,Z 283.45,A -85,B 0,C 180,E1 -4137.755,E2 -4137.755} C_VEL
LIN {X 0,Y 538.167,Z 283.443,A -85,B 0,C 180,E1 -4140.748,E2 -4140.748} C_VEL
LIN {X 0,Y 538.124,Z 283.45,A -85,B 0,C 180,E1 -4142.995,E2 -4142.995} C_VEL
LIN {X 0,Y 538.098,Z 283.455,A -85,B 0,C 180,E1 -4145.998,E2 -4145.998} C_VEL
LIN {X 0,Y 538.046,Z 283.458,A -85,B 0,C 180,E1 -4149.018,E2 -4149.018} C_VEL
LIN {X 0,Y 538.051,Z 283.462,A -85,B 0,C 180,E1 -4152.063,E2 -4152.063} C_VEL
LIN {X 0,Y 538.028,Z 283.461,A -85,B 0,C 180,E1 -4155.144,E2 -4155.144} C_VEL
LIN {X 0,Y 538.003,Z 283.467,A -85,B 0,C 180,E1 -4158.271,E2 -4158.271} C_VEL
LIN {X 0,Y 538.021,Z 283.462,A -85,B 0,C 180,E1 -4160.652,E2 -4160.652} C_VEL
LIN {X 0,Y 537.997,Z 283.471,A -85,B 0,C 180,E1 -4163.878,E2 -4163.878} C_VEL
LIN {X 0,Y 537.973,Z 283.472,A -85,B 0,C 180,E1 -4166.37,E2 -4166.37} C_VEL
LIN {X 0,Y 537.984,Z 283.466,A -85,B 0,C 180,E1 -4168.926,E2 -4168.926} C_VEL
LIN {X 0,Y 538.002,Z 283.467,A -85,B 0,C 180,E1 -4171.887,E2 -4171.887} C_VEL
LIN {X 0,Y 537.988,Z 283.47,A -85,B 0,C 180,E1 -4174.615,E2 -4174.615} C_VEL
LIN {X 0,Y 537.969,Z 283.47,A -85,B 0,C 180,E1 -4177.88,E2 -4177.88} C_VEL
LIN {X 0,Y 537.957,Z 283.47,A -85,B 0,C 180,E1 -4180.241,E2 -4180.241} C_VEL
LIN {X 0,Y 537.305,Z 283.555,A -85,B 0,C 180,E1 -4180.867,E2 -4180.867} C_VEL
LIN {X 0,Y 534.456,Z 283.907,A -85,B 0,C 180,E1 -4181.881,E2 -4181.881} C_VEL
LIN {X 0,Y 532.039,Z 284.213,A -85,B 0,C 180,E1 -4182.698,E2 -4182.698} C_VEL
LIN {X 0,Y 531,Z 284.336,A -85,B 0,C 180,E1 -4183.329,E2 -4183.329} C_VEL
LIN {X 0,Y 530.915,Z 284.346,A -85,B 0,C 180,E1 -4183.543,E2 -4183.543} C_VEL
LIN {X 0,Y 530.958,Z 284.34,A -85,B 0,C 180,E1 -4185.624,E2 -4185.624} C_VEL
LIN {X 0,Y 530.905,Z 284.356,A -85,B 0,C 180,E1 -4188.556,E2 -4188.556} C_VEL
LIN {X 0,Y 530.912,Z 284.347,A -85,B 0,C 180,E1 -4191.525,E2 -4191.525} C_VEL
LIN {X 0,Y 530.904,Z 284.351,A -85,B 0,C 180,E1 -4194.376,E2 -4194.376} C_VEL
LIN {X 0,Y 530.936,Z 284.349,A -85,B 0,C 180,E1 -4197.131,E2 -4197.131} C_VEL
LIN {X 0,Y 530.928,Z 284.344,A -85,B 0,C 180,E1 -4199.8,E2 -4199.8} C_VEL
LIN {X 0,Y 530.957,Z 284.343,A -85,B 0,C 180,E1 -4202.48,E2 -4202.48} C_VEL
LIN {X 0,Y 530.949,Z 284.342,A -85,B 0,C 180,E1 -4205.773,E2 -4205.773} C_VEL
LIN {X 0,Y 530.999,Z 284.344,A -85,B 0,C 180,E1 -4209.061,E2 -4209.061} C_VEL
LIN {X 0,Y 530.964,Z 284.345,A -85,B 0,C 180,E1 -4211.477,E2 -4211.477} C_VEL
LIN {X 0,Y 530.989,Z 284.338,A -85,B 0,C 180,E1 -4214.649,E2 -4214.649} C_VEL
LIN {X 0,Y 531.023,Z 284.336,A -85,B 0,C 180,E1 -4217.773,E2 -4217.773} C_VEL
LIN {X 0,Y 530.965,Z 284.341,A -85,B 0,C 180,E1 -4220.09,E2 -4220.09} C_VEL
LIN {X 0,Y 531.017,Z 284.338,A -85,B 0,C 180,E1 -4223.157,E2 -4223.157} C_VEL
LIN {X 0,Y 530.987,Z 284.346,A -85,B 0,C 180,E1 -4225.443,E2 -4225.443} C_VEL
LIN {X 0,Y 531.136,Z 284.326,A -85,B 0,C 180,E1 -4227.723,E2 -4227.723} C_VEL
LIN {X 0,Y 531.131,Z 284.323,A -85,B 0,C 180,E1 -4229.998,E2 -4229.998} C_VEL
LIN {X 0,Y 531.06,Z 284.329,A -85,B 0,C 180,E1 -4233.032,E2 -4233.032} C_VEL
LIN {X 0,Y 531.048,Z 284.336,A -85,B 0,C 180,E1 -4236.075,E2 -4236.075} C_VEL
LIN {X 0,Y 531.01,Z 284.337,A -85,B 0,C 180,E1 -4239.135,E2 -4239.135} C_VEL
LIN {X 0,Y 531.067,Z 284.417,A -85,B 0,C 180,E1 -4242.415,E2 -4242.415} C_VEL
LIN {X 0,Y 531.462,Z 290.395,A -85,B 0,C 180,E1 -4243.572,E2 -4243.572} C_VEL
LIN {X 0,Y 531.253,Z 304.945,A -85,B 0,C 180,E1 -4246.323,E2 -4246.323} C_VEL
LIN {X 0,Y 531.217,Z 309.171,A -85,B 0,C 180,E1 -4247.113,E2 -4247.113} C_VEL
LIN {X 0,Y 532.793,Z 317.943,A -85,B 0,C 180,E1 -4247.279,E2 -4247.279} C_VEL
LIN {X 0,Y 532.396,Z 415.362,A -85,B 0,C 180,E1 -4248.616,E2 -4248.616} C_VEL
LIN {X 0,Y 532.266,Z 428.487,A -85,B 0,C 180,E1 -4248.945,E2 -4248.945} C_VEL
LIN {X 0,Y 532.046,Z 441.393,A -85,B 0,C 180,E1 -4249.429,E2 -4249.429} C_VEL
LIN {X 0,Y 531.803,Z 452.503,A -85,B 0,C 180,E1 -4249.992,E2 -4249.992} C_VEL
LIN {X 0,Y 531.536,Z 463.319,A -85,B 0,C 180,E1 -4250.693,E2 -4250.693} C_VEL
LIN {X 0,Y 531.301,Z 473.672,A -85,B 0,C 180,E1 -4251.531,E2 -4251.531} C_VEL
LIN {X 0,Y 531.058,Z 483.98,A -85,B 0,C 180,E1 -4252.564,E2 -4252.564} C_VEL
LIN {X 0,Y 530.844,Z 492.97,A -85,B 0,C 180,E1 -4253.696,E2 -4253.696} C_VEL
LIN {X 0,Y 530.677,Z 500.412,A -85,B 0,C 180,E1 -4254.86,E2 -4254.86} C_VEL
LIN {X 0,Y 530.59,Z 505.847,A -85,B 0,C 180,E1 -4255.915,E2 -4255.915} C_VEL
LIN {X 0,Y 530.521,Z 510.691,A -85,B 0,C 180,E1 -4257.093,E2 -4257.093} C_VEL
LIN {X 0,Y 530.418,Z 514.933,A -85,B 0,C 180,E1 -4258.484,E2 -4258.484} C_VEL
LIN {X 0,Y 530.389,Z 516.806,A -85,B 0,C 180,E1 -4259.354,E2 -4259.354} C_VEL
LIN {X 0,Y 530.382,Z 518.511,A -85,B 0,C 180,E1 -4260.536,E2 -4260.536} C_VEL
LIN {X 0,Y 530.356,Z 519.312,A -85,B 0,C 180,E1 -4262.004,E2 -4262.004} C_VEL
LIN {X 0,Y 530.351,Z 518.676,A -85,B 0,C 180,E1 -4263.399,E2 -4263.399} C_VEL
LIN {X 0,Y 530.371,Z 516.77,A -85,B 0,C 180,E1 -4264.758,E2 -4264.758} C_VEL
LIN {X 0,Y 530.468,Z 513.648,A -85,B 0,C 180,E1 -4266.082,E2 -4266.082} C_VEL
LIN {X 0,Y 530.544,Z 509.349,A -85,B 0,C 180,E1 -4267.363,E2 -4267.363} C_VEL
LIN {X 0,Y 530.626,Z 503.789,A -85,B 0,C 180,E1 -4268.607,E2 -4268.607} C_VEL
LIN {X 0,Y 530.773,Z 496.818,A -85,B 0,C 180,E1 -4269.827,E2 -4269.827} C_VEL
LIN {X 0,Y 530.956,Z 488.287,A -85,B 0,C 180,E1 -4271.02,E2 -4271.02} C_VEL
LIN {X 0,Y 531.194,Z 479.001,A -85,B 0,C 180,E1 -4272.056,E2 -4272.056} C_VEL
LIN {X 0,Y 531.465,Z 468.215,A -85,B 0,C 180,E1 -4273.026,E2 -4273.026} C_VEL
LIN {X 0,Y 531.664,Z 457.34,A -85,B 0,C 180,E1 -4273.808,E2 -4273.808} C_VEL
LIN {X 0,Y 531.969,Z 445.153,A -85,B 0,C 180,E1 -4274.487,E2 -4274.487} C_VEL
LIN {X 0,Y 532.171,Z 433.836,A -85,B 0,C 180,E1 -4274.966,E2 -4274.966} C_VEL
LIN {X 0,Y 532.359,Z 421.101,A -85,B 0,C 180,E1 -4275.352,E2 -4275.352} C_VEL
LIN {X 0,Y 532.485,Z 407.706,A -85,B 0,C 180,E1 -4275.592,E2 -4275.592} C_VEL
LIN {X 0,Y 532.696,Z 317.442,A -85,B 0,C 180,E1 -4276.821,E2 -4276.821} C_VEL
LIN {X 0,Y 531.184,Z 308.736,A -85,B 0,C 180,E1 -4276.992,E2 -4276.992} C_VEL
LIN {X 0,Y 531.251,Z 294.056,A -85,B 0,C 180,E1 -4279.592,E2 -4279.592} C_VEL
LIN {X 0,Y 531.086,Z 284.795,A -85,B 0,C 180,E1 -4281.194,E2 -4281.194} C_VEL
LIN {X 0,Y 531.031,Z 284.338,A -85,B 0,C 180,E1 -4281.329,E2 -4281.329} C_VEL
LIN {X 0,Y 530.943,Z 284.352,A -85,B 0,C 180,E1 -4284.379,E2 -4284.379} C_VEL
LIN {X 0,Y 530.933,Z 284.346,A -85,B 0,C 180,E1 -4287.131,E2 -4287.131} C_VEL
LIN {X 0,Y 530.941,Z 284.347,A -85,B 0,C 180,E1 -4289.801,E2 -4289.801} C_VEL
LIN {X 0,Y 530.971,Z 284.349,A -85,B 0,C 180,E1 -4292.463,E2 -4292.463} C_VEL
LIN {X 0,Y 530.969,Z 284.345,A -85,B 0,C 180,E1 -4294.94,E2 -4294.94} C_VEL
LIN {X 0,Y 530.92,Z 284.354,A -85,B 0,C 180,E1 -4298.244,E2 -4298.244} C_VEL
LIN {X 0,Y 530.944,Z 284.35,A -85,B 0,C 180,E1 -4300.675,E2 -4300.675} C_VEL
LIN {X 0,Y 530.932,Z 284.347,A -85,B 0,C 180,E1 -4303.069,E2 -4303.069} C_VEL
LIN {X 0,Y 530.964,Z 284.341,A -85,B 0,C 180,E1 -4305.434,E2 -4305.434} C_VEL
LIN {X 0,Y 530.992,Z 284.345,A -85,B 0,C 180,E1 -4308.549,E2 -4308.549} C_VEL
LIN {X 0,Y 531.002,Z 284.336,A -85,B 0,C 180,E1 -4311.629,E2 -4311.629} C_VEL
LIN {X 0,Y 531.086,Z 284.334,A -85,B 0,C 180,E1 -4314.685,E2 -4314.685} C_VEL
LIN {X 0,Y 531.079,Z 284.326,A -85,B 0,C 180,E1 -4317.725,E2 -4317.725} C_VEL
LIN {X 0,Y 531.106,Z 284.328,A -85,B 0,C 180,E1 -4320.758,E2 -4320.758} C_VEL
LIN {X 0,Y 531.061,Z 284.334,A -85,B 0,C 180,E1 -4323.034,E2 -4323.034} C_VEL
LIN {X 0,Y 531.033,Z 284.332,A -85,B 0,C 180,E1 -4326.078,E2 -4326.078} C_VEL
LIN {X 0,Y 530.991,Z 284.346,A -85,B 0,C 180,E1 -4329.139,E2 -4329.139} C_VEL
LIN {X 0,Y 531.012,Z 284.333,A -85,B 0,C 180,E1 -4331.682,E2 -4331.682} C_VEL
LIN {X 0,Y 530.994,Z 284.343,A -85,B 0,C 180,E1 -4334.965,E2 -4334.965} C_VEL
LIN {X 0,Y 530.967,Z 284.341,A -85,B 0,C 180,E1 -4337.724,E2 -4337.724} C_VEL
LIN {X 0,Y 530.962,Z 284.343,A -85,B 0,C 180,E1 -4340.94,E2 -4340.94} C_VEL
LIN {X 0,Y 530.979,Z 284.336,A -85,B 0,C 180,E1 -4344.052,E2 -4344.052} C_VEL
LIN {X 0,Y 530.978,Z 284.339,A -85,B 0,C 180,E1 -4346.745,E2 -4346.745} C_VEL
LIN {X 0,Y 530.963,Z 284.347,A -85,B 0,C 180,E1 -4349.324,E2 -4349.324} C_VEL
LIN {X 0,Y 530.945,Z 284.343,A -85,B 0,C 180,E1 -4352.108,E2 -4352.108} C_VEL
LIN {X 0,Y 530.954,Z 284.342,A -85,B 0,C 180,E1 -4354.859,E2 -4354.859} C_VEL
LIN {X 0,Y 530.946,Z 284.352,A -85,B 0,C 180,E1 -4357.509,E2 -4357.509} C_VEL
LIN {X 0,Y 531.008,Z 284.336,A -85,B 0,C 180,E1 -4360.431,E2 -4360.431} C_VEL
LIN {X 0,Y 530.935,Z 284.352,A -85,B 0,C 180,E1 -4363.498,E2 -4363.498} C_VEL
LIN {X 0,Y 530.938,Z 284.346,A -85,B 0,C 180,E1 -4366.51,E2 -4366.51} C_VEL
LIN {X 0,Y 531.001,Z 284.344,A -85,B 0,C 180,E1 -4369.575,E2 -4369.575} C_VEL
LIN {X 0,Y 530.954,Z 284.343,A -85,B 0,C 180,E1 -4372.579,E2 -4372.579} C_VEL
LIN {X 0,Y 530.983,Z 284.341,A -85,B 0,C 180,E1 -4375.315,E2 -4375.315} C_VEL
LIN {X 0,Y 530.965,Z 284.35,A -85,B 0,C 180,E1 -4378.037,E2 -4378.037} C_VEL
LIN {X 0,Y 530.991,Z 284.34,A -85,B 0,C 180,E1 -4380.874,E2 -4380.874} C_VEL
LIN {X 0,Y 530.998,Z 284.339,A -85,B 0,C 180,E1 -4383.261,E2 -4383.261} C_VEL
LIN {X 0,Y 531.016,Z 284.436,A -85,B 0,C 180,E1 -4385.73,E2 -4385.73} C_VEL
LIN {X 0,Y 532.289,Z 291.544,A -85,B 0,C 180,E1 -4386.876,E2 -4386.876} C_VEL
LIN {X 0,Y 531.905,Z 312.853,A -85,B 0,C 180,E1 -4390.113,E2 -4390.113} C_VEL
LIN {X 0,Y 531.473,Z 332.675,A -85,B 0,C 180,E1 -4393.091,E2 -4393.091} C_VEL
LIN {X 0,Y 531.295,Z 346.08,A -85,B 0,C 180,E1 -4395.051,E2 -4395.051} C_VEL
LIN {X 0,Y 532.8,Z 357.19,A -85,B 0,C 180,E1 -4395.247,E2 -4395.247} C_VEL
LIN {X 0,Y 532.374,Z 454.114,A -85,B 0,C 180,E1 -4396.573,E2 -4396.573} C_VEL
LIN {X 0,Y 532.186,Z 467.46,A -85,B 0,C 180,E1 -4396.909,E2 -4396.909} C_VEL
LIN {X 0,Y 531.908,Z 480.796,A -85,B 0,C 180,E1 -4397.411,E2 -4397.411} C_VEL
LIN {X 0,Y 531.784,Z 491.786,A -85,B 0,C 180,E1 -4397.977,E2 -4397.977} C_VEL
LIN {X 0,Y 531.505,Z 503.628,A -85,B 0,C 180,E1 -4398.756,E2 -4398.756} C_VEL
LIN {X 0,Y 531.201,Z 514.101,A -85,B 0,C 180,E1 -4399.618,E2 -4399.618} C_VEL
LIN {X 0,Y 531.016,Z 522.667,A -85,B 0,C 180,E1 -4400.481,E2 -4400.481} C_VEL
LIN {X 0,Y 530.878,Z 530.571,A -85,B 0,C 180,E1 -4401.438,E2 -4401.438} C_VEL
LIN {X 0,Y 530.671,Z 538.286,A -85,B 0,C 180,E1 -4402.584,E2 -4402.584} C_VEL
LIN {X 0,Y 530.59,Z 545.4,A -85,B 0,C 180,E1 -4403.92,E2 -4403.92} C_VEL
LIN {X 0,Y 530.458,Z 550.13,A -85,B 0,C 180,E1 -4405.063,E2 -4405.063} C_VEL
LIN {X 0,Y 530.515,Z 553.748,A -85,B 0,C 180,E1 -4406.205,E2 -4406.205} C_VEL
LIN {X 0,Y 530.456,Z 555.61,A -85,B 0,C 180,E1 -4406.965,E2 -4406.965} C_VEL
LIN {X 0,Y 530.41,Z 557.006,A -85,B 0,C 180,E1 -4407.724,E2 -4407.724} C_VEL
LIN {X 0,Y 530.344,Z 558.61,A -85,B 0,C 180,E1 -4409.243,E2 -4409.243} C_VEL
LIN {X 0,Y 530.345,Z 558.826,A -85,B 0,C 180,E1 -4410.002,E2 -4410.002} C_VEL
LIN {X 0,Y 530.361,Z 558,A -85,B 0,C 180,E1 -4411.521,E2 -4411.521} C_VEL
LIN {X 0,Y 530.411,Z 557.005,A -85,B 0,C 180,E1 -4412.28,E2 -4412.28} C_VEL
LIN {X 0,Y 530.457,Z 555.607,A -85,B 0,C 180,E1 -4413.04,E2 -4413.04} C_VEL
LIN {X 0,Y 530.523,Z 552.668,A -85,B 0,C 180,E1 -4414.18,E2 -4414.18} C_VEL
LIN {X 0,Y 530.525,Z 548.684,A -85,B 0,C 180,E1 -4415.323,E2 -4415.323} C_VEL
LIN {X 0,Y 530.567,Z 543.119,A -85,B 0,C 180,E1 -4416.552,E2 -4416.552} C_VEL
LIN {X 0,Y 530.698,Z 537.106,A -85,B 0,C 180,E1 -4417.612,E2 -4417.612} C_VEL
LIN {X 0,Y 530.867,Z 529.058,A -85,B 0,C 180,E1 -4418.759,E2 -4418.759} C_VEL
LIN {X 0,Y 531.079,Z 520.856,A -85,B 0,C 180,E1 -4419.716,E2 -4419.716} C_VEL
LIN {X 0,Y 531.317,Z 510.854,A -85,B 0,C 180,E1 -4420.674,E2 -4420.674} C_VEL
LIN {X 0,Y 531.603,Z 500.984,A -85,B 0,C 180,E1 -4421.44,E2 -4421.44} C_VEL
LIN {X 0,Y 531.762,Z 490.455,A -85,B 0,C 180,E1 -4422.102,E2 -4422.102} C_VEL
LIN {X 0,Y 531.998,Z 477.337,A -85,B 0,C 180,E1 -4422.737,E2 -4422.737} C_VEL
LIN {X 0,Y 532.209,Z 464.184,A -85,B 0,C 180,E1 -4423.193,E2 -4423.193} C_VEL
LIN {X 0,Y 532.409,Z 451.002,A -85,B 0,C 180,E1 -4423.479,E2 -4423.479} C_VEL
LIN {X 0,Y 532.721,Z 355.329,A -85,B 0,C 180,E1 -4424.783,E2 -4424.783} C_VEL
LIN {X 0,Y 531.317,Z 345.912,A -85,B 0,C 180,E1 -4424.968,E2 -4424.968} C_VEL
LIN {X 0,Y 531.722,Z 324.991,A -85,B 0,C 180,E1 -4428.119,E2 -4428.119} C_VEL
LIN {X 0,Y 532.047,Z 306.752,A -85,B 0,C 180,E1 -4430.896,E2 -4430.896} C_VEL
LIN {X 0,Y 532.407,Z 292.366,A -85,B 0,C 180,E1 -4433.124,E2 -4433.124} C_VEL
LIN {X 0,Y 530.997,Z 284.342,A -85,B 0,C 180,E1 -4434.485,E2 -4434.485} C_VEL
LIN {X 0,Y 531.014,Z 284.34,A -85,B 0,C 180,E1 -4437.532,E2 -4437.532} C_VEL
LIN {X 0,Y 530.978,Z 284.341,A -85,B 0,C 180,E1 -4440.645,E2 -4440.645} C_VEL
LIN {X 0,Y 530.99,Z 284.34,A -85,B 0,C 180,E1 -4443.773,E2 -4443.773} C_VEL
LIN {X 0,Y 530.957,Z 284.345,A -85,B 0,C 180,E1 -4446.559,E2 -4446.559} C_VEL
LIN {X 0,Y 530.986,Z 284.337,A -85,B 0,C 180,E1 -4449.443,E2 -4449.443} C_VEL
LIN {X 0,Y 530.979,Z 284.346,A -85,B 0,C 180,E1 -4452.456,E2 -4452.456} C_VEL
LIN {X 0,Y 530.975,Z 284.339,A -85,B 0,C 180,E1 -4455.622,E2 -4455.622} C_VEL
LIN {X 0,Y 530.998,Z 284.345,A -85,B 0,C 180,E1 -4458.565,E2 -4458.565} C_VEL
LIN {X 0,Y 530.954,Z 284.341,A -85,B 0,C 180,E1 -4461.529,E2 -4461.529} C_VEL
LIN {X 0,Y 530.971,Z 284.345,A -85,B 0,C 180,E1 -4464.381,E2 -4464.381} C_VEL
LIN {X 0,Y 530.966,Z 284.343,A -85,B 0,C 180,E1 -4467.133,E2 -4467.133} C_VEL
LIN {X 0,Y 530.98,Z 284.338,A -85,B 0,C 180,E1 -4469.804,E2 -4469.804} C_VEL
LIN {X 0,Y 531.009,Z 284.338,A -85,B 0,C 180,E1 -4472.466,E2 -4472.466} C_VEL
LIN {X 0,Y 530.999,Z 284.345,A -85,B 0,C 180,E1 -4474.942,E2 -4474.942} C_VEL
LIN {X 0,Y 530.961,Z 284.341,A -85,B 0,C 180,E1 -4478.246,E2 -4478.246} C_VEL
LIN {X 0,Y 530.984,Z 284.342,A -85,B 0,C 180,E1 -4480.677,E2 -4480.677} C_VEL
LIN {X 0,Y 530.974,Z 284.349,A -85,B 0,C 180,E1 -4483.071,E2 -4483.071} C_VEL
LIN {X 0,Y 531.007,Z 284.34,A -85,B 0,C 180,E1 -4485.435,E2 -4485.435} C_VEL
LIN {X 0,Y 531.027,Z 284.333,A -85,B 0,C 180,E1 -4488.549,E2 -4488.549} C_VEL
LIN {X 0,Y 531.042,Z 284.335,A -85,B 0,C 180,E1 -4491.629,E2 -4491.629} C_VEL
LIN {X 0,Y 531.11,Z 284.323,A -85,B 0,C 180,E1 -4494.685,E2 -4494.685} C_VEL
LIN {X 0,Y 531.122,Z 284.325,A -85,B 0,C 180,E1 -4497.725,E2 -4497.725} C_VEL
LIN {X 0,Y 531.138,Z 284.319,A -85,B 0,C 180,E1 -4500.758,E2 -4500.758} C_VEL
LIN {X 0,Y 531.091,Z 284.326,A -85,B 0,C 180,E1 -4503.034,E2 -4503.034} C_VEL
LIN {X 0,Y 531.053,Z 284.332,A -85,B 0,C 180,E1 -4506.077,E2 -4506.077} C_VEL
LIN {X 0,Y 531.009,Z 284.336,A -85,B 0,C 180,E1 -4509.139,E2 -4509.139} C_VEL
LIN {X 0,Y 531.014,Z 284.337,A -85,B 0,C 180,E1 -4512.226,E2 -4512.226} C_VEL
LIN {X 0,Y 530.977,Z 284.341,A -85,B 0,C 180,E1 -4515.35,E2 -4515.35} C_VEL
LIN {X 0,Y 530.964,Z 284.341,A -85,B 0,C 180,E1 -4518.522,E2 -4518.522} C_VEL
LIN {X 0,Y 530.983,Z 284.337,A -85,B 0,C 180,E1 -4520.939,E2 -4520.939} C_VEL
LIN {X 0,Y 530.942,Z 284.35,A -85,B 0,C 180,E1 -4524.226,E2 -4524.226} C_VEL
LIN {X 0,Y 530.936,Z 284.345,A -85,B 0,C 180,E1 -4526.748,E2 -4526.748} C_VEL
LIN {X 0,Y 530.952,Z 284.341,A -85,B 0,C 180,E1 -4529.325,E2 -4529.325} C_VEL
LIN {X 0,Y 530.956,Z 284.348,A -85,B 0,C 180,E1 -4532.1,E2 -4532.1} C_VEL
LIN {X 0,Y 530.949,Z 284.344,A -85,B 0,C 180,E1 -4534.849,E2 -4534.849} C_VEL
LIN {X 0,Y 530.922,Z 284.345,A -85,B 0,C 180,E1 -4537.512,E2 -4537.512} C_VEL
LIN {X 0,Y 530.926,Z 284.355,A -85,B 0,C 180,E1 -4540.438,E2 -4540.438} C_VEL
LIN {X 0,Y 530.915,Z 284.346,A -85,B 0,C 180,E1 -4543.543,E2 -4543.543} C_VEL
LIN {X 0,Y 530.253,Z 284.434,A -85,B 0,C 180,E1 -4544.177,E2 -4544.177} C_VEL
LIN {X 0,Y 527.413,Z 284.792,A -85,B 0,C 180,E1 -4545.206,E2 -4545.206} C_VEL
LIN {X 0,Y 525.003,Z 285.094,A -85,B 0,C 180,E1 -4546.034,E2 -4546.034} C_VEL
LIN {X 0,Y 523.957,Z 285.221,A -85,B 0,C 180,E1 -4546.674,E2 -4546.674} C_VEL
LIN {X 0,Y 523.865,Z 285.229,A -85,B 0,C 180,E1 -4546.891,E2 -4546.891} C_VEL
LIN {X 0,Y 523.861,Z 285.225,A -85,B 0,C 180,E1 -4549.913,E2 -4549.913} C_VEL
LIN {X 0,Y 523.846,Z 285.235,A -85,B 0,C 180,E1 -4552.863,E2 -4552.863} C_VEL
LIN {X 0,Y 523.866,Z 285.224,A -85,B 0,C 180,E1 -4555.704,E2 -4555.704} C_VEL
LIN {X 0,Y 523.905,Z 285.222,A -85,B 0,C 180,E1 -4558.454,E2 -4558.454} C_VEL
LIN {X 0,Y 523.873,Z 285.23,A -85,B 0,C 180,E1 -4561.121,E2 -4561.121} C_VEL
LIN {X 0,Y 523.88,Z 285.222,A -85,B 0,C 180,E1 -4564.004,E2 -4564.004} C_VEL
LIN {X 0,Y 523.91,Z 285.219,A -85,B 0,C 180,E1 -4566.269,E2 -4566.269} C_VEL
LIN {X 0,Y 523.947,Z 285.218,A -85,B 0,C 180,E1 -4568.766,E2 -4568.766} C_VEL
LIN {X 0,Y 523.925,Z 285.226,A -85,B 0,C 180,E1 -4571.218,E2 -4571.218} C_VEL
LIN {X 0,Y 523.895,Z 285.224,A -85,B 0,C 180,E1 -4573.636,E2 -4573.636} C_VEL
LIN {X 0,Y 523.921,Z 285.218,A -85,B 0,C 180,E1 -4576.026,E2 -4576.026} C_VEL
LIN {X 0,Y 524.019,Z 285.205,A -85,B 0,C 180,E1 -4578.393,E2 -4578.393} C_VEL
LIN {X 0,Y 523.95,Z 285.222,A -85,B 0,C 180,E1 -4581.513,E2 -4581.513} C_VEL
LIN {X 0,Y 524.037,Z 285.203,A -85,B 0,C 180,E1 -4584.611,E2 -4584.611} C_VEL
LIN {X 0,Y 524.107,Z 285.202,A -85,B 0,C 180,E1 -4587.692,E2 -4587.692} C_VEL
LIN {X 0,Y 524.099,Z 285.199,A -85,B 0,C 180,E1 -4589.998,E2 -4589.998} C_VEL
LIN {X 0,Y 524.106,Z 285.195,A -85,B 0,C 180,E1 -4592.303,E2 -4592.303} C_VEL
LIN {X 0,Y 524.009,Z 285.212,A -85,B 0,C 180,E1 -4596.157,E2 -4596.157} C_VEL
LIN {X 0,Y 523.979,Z 285.214,A -85,B 0,C 180,E1 -4599.259,E2 -4599.259} C_VEL
LIN {X 0,Y 524.006,Z 285.234,A -85,B 0,C 180,E1 -4602.29,E2 -4602.29} C_VEL
LIN {X 0,Y 524.479,Z 290.704,A -85,B 0,C 180,E1 -4603.361,E2 -4603.361} C_VEL
LIN {X 0,Y 524.264,Z 305.312,A -85,B 0,C 180,E1 -4606.147,E2 -4606.147} C_VEL
LIN {X 0,Y 524.208,Z 309.3,A -85,B 0,C 180,E1 -4606.9,E2 -4606.9} C_VEL
LIN {X 0,Y 525.947,Z 318.815,A -85,B 0,C 180,E1 -4607.092,E2 -4607.092} C_VEL
LIN {X 0,Y 525.486,Z 416.635,A -85,B 0,C 180,E1 -4608.46,E2 -4608.46} C_VEL
LIN {X 0,Y 525.354,Z 429.56,A -85,B 0,C 180,E1 -4608.799,E2 -4608.799} C_VEL
LIN {X 0,Y 525.118,Z 442.258,A -85,B 0,C 180,E1 -4609.29,E2 -4609.29} C_VEL
LIN {X 0,Y 524.869,Z 453.198,A -85,B 0,C 180,E1 -4609.859,E2 -4609.859} C_VEL
LIN {X 0,Y 524.561,Z 464.156,A -85,B 0,C 180,E1 -4610.587,E2 -4610.587} C_VEL
LIN {X 0,Y 524.298,Z 475.367,A -85,B 0,C 180,E1 -4611.523,E2 -4611.523} C_VEL
LIN {X 0,Y 524.023,Z 485.114,A -85,B 0,C 180,E1 -4612.541,E2 -4612.541} C_VEL
LIN {X 0,Y 523.804,Z 494.237,A -85,B 0,C 180,E1 -4613.731,E2 -4613.731} C_VEL
LIN {X 0,Y 523.626,Z 500.837,A -85,B 0,C 180,E1 -4614.794,E2 -4614.794} C_VEL
LIN {X 0,Y 523.528,Z 506.493,A -85,B 0,C 180,E1 -4615.917,E2 -4615.917} C_VEL
LIN {X 0,Y 523.441,Z 511.424,A -85,B 0,C 180,E1 -4617.157,E2 -4617.157} C_VEL
LIN {X 0,Y 523.339,Z 515.263,A -85,B 0,C 180,E1 -4618.467,E2 -4618.467} C_VEL
LIN {X 0,Y 523.307,Z 517.86,A -85,B 0,C 180,E1 -4619.791,E2 -4619.791} C_VEL
LIN {X 0,Y 523.284,Z 518.998,A -85,B 0,C 180,E1 -4620.733,E2 -4620.733} C_VEL
LIN {X 0,Y 523.251,Z 519.554,A -85,B 0,C 180,E1 -4622.201,E2 -4622.201} C_VEL
LIN {X 0,Y 523.27,Z 518.731,A -85,B 0,C 180,E1 -4623.621,E2 -4623.621} C_VEL
LIN {X 0,Y 523.282,Z 516.674,A -85,B 0,C 180,E1 -4624.988,E2 -4624.988} C_VEL
LIN {X 0,Y 523.387,Z 513.395,A -85,B 0,C 180,E1 -4626.324,E2 -4626.324} C_VEL
LIN {X 0,Y 523.486,Z 508.881,A -85,B 0,C 180,E1 -4627.618,E2 -4627.618} C_VEL
LIN {X 0,Y 523.566,Z 503.143,A -85,B 0,C 180,E1 -4628.871,E2 -4628.871} C_VEL
LIN {X 0,Y 523.77,Z 495.964,A -85,B 0,C 180,E1 -4630.108,E2 -4630.108} C_VEL
LIN {X 0,Y 523.981,Z 487.125,A -85,B 0,C 180,E1 -4631.313,E2 -4631.313} C_VEL
LIN {X 0,Y 524.215,Z 478.197,A -85,B 0,C 180,E1 -4632.296,E2 -4632.296} C_VEL
LIN {X 0,Y 524.493,Z 467.587,A -85,B 0,C 180,E1 -4633.246,E2 -4633.246} C_VEL
LIN {X 0,Y 524.76,Z 456.095,A -85,B 0,C 180,E1 -4634.057,E2 -4634.057} C_VEL
LIN {X 0,Y 525.07,Z 443.494,A -85,B 0,C 180,E1 -4634.746,E2 -4634.746} C_VEL
LIN {X 0,Y 525.346,Z 430.891,A -85,B 0,C 180,E1 -4635.25,E2 -4635.25} C_VEL
LIN {X 0,Y 525.508,Z 417.669,A -85,B 0,C 180,E1 -4635.608,E2 -4635.608} C_VEL
LIN {X 0,Y 525.651,Z 387.424,A -85,B 0,C 180,E1 -4636.055,E2 -4636.055} C_VEL
LIN {X 0,Y 525.886,Z 318.366,A -85,B 0,C 180,E1 -4637.008,E2 -4637.008} C_VEL
LIN {X 0,Y 524.194,Z 308.969,A -85,B 0,C 180,E1 -4637.197,E2 -4637.197} C_VEL
LIN {X 0,Y 524.246,Z 293.338,A -85,B 0,C 180,E1 -4639.948,E2 -4639.948} C_VEL
LIN {X 0,Y 524.013,Z 285.263,A -85,B 0,C 180,E1 -4641.35,E2 -4641.35} C_VEL
LIN {X 0,Y 523.899,Z 285.224,A -85,B 0,C 180,E1 -4644.905,E2 -4644.905} C_VEL
LIN {X 0,Y 523.9,Z 285.223,A -85,B 0,C 180,E1 -4647.675,E2 -4647.675} C_VEL
LIN {X 0,Y 523.924,Z 285.223,A -85,B 0,C 180,E1 -4650.67,E2 -4650.67} C_VEL
LIN {X 0,Y 523.933,Z 285.22,A -85,B 0,C 180,E1 -4653.726,E2 -4653.726} C_VEL
LIN {X 0,Y 523.887,Z 285.232,A -85,B 0,C 180,E1 -4656.268,E2 -4656.268} C_VEL
LIN {X 0,Y 523.894,Z 285.228,A -85,B 0,C 180,E1 -4658.764,E2 -4658.764} C_VEL
LIN {X 0,Y 523.901,Z 285.222,A -85,B 0,C 180,E1 -4661.219,E2 -4661.219} C_VEL
LIN {X 0,Y 523.883,Z 285.223,A -85,B 0,C 180,E1 -4663.637,E2 -4663.637} C_VEL
LIN {X 0,Y 523.886,Z 285.224,A -85,B 0,C 180,E1 -4666.026,E2 -4666.026} C_VEL
LIN {X 0,Y 523.957,Z 285.219,A -85,B 0,C 180,E1 -4668.393,E2 -4668.393} C_VEL
LIN {X 0,Y 523.95,Z 285.214,A -85,B 0,C 180,E1 -4671.515,E2 -4671.515} C_VEL
LIN {X 0,Y 524.043,Z 285.21,A -85,B 0,C 180,E1 -4674.613,E2 -4674.613} C_VEL
LIN {X 0,Y 524.052,Z 285.201,A -85,B 0,C 180,E1 -4677.694,E2 -4677.694} C_VEL
LIN {X 0,Y 524.075,Z 285.204,A -85,B 0,C 180,E1 -4680.768,E2 -4680.768} C_VEL
LIN {X 0,Y 524.027,Z 285.209,A -85,B 0,C 180,E1 -4683.075,E2 -4683.075} C_VEL
LIN {X 0,Y 523.994,Z 285.209,A -85,B 0,C 180,E1 -4686.16,E2 -4686.16} C_VEL
LIN {X 0,Y 523.959,Z 285.219,A -85,B 0,C 180,E1 -4689.263,E2 -4689.263} C_VEL
LIN {X 0,Y 523.97,Z 285.21,A -85,B 0,C 180,E1 -4691.753,E2 -4691.753} C_VEL
LIN {X 0,Y 523.953,Z 285.222,A -85,B 0,C 180,E1 -4695.06,E2 -4695.06} C_VEL
LIN {X 0,Y 523.916,Z 285.218,A -85,B 0,C 180,E1 -4697.971,E2 -4697.971} C_VEL
LIN {X 0,Y 523.925,Z 285.215,A -85,B 0,C 180,E1 -4700.412,E2 -4700.412} C_VEL
LIN {X 0,Y 523.922,Z 285.22,A -85,B 0,C 180,E1 -4702.893,E2 -4702.893} C_VEL
LIN {X 0,Y 523.938,Z 285.224,A -85,B 0,C 180,E1 -4705.42,E2 -4705.42} C_VEL
LIN {X 0,Y 523.928,Z 285.216,A -85,B 0,C 180,E1 -4708.001,E2 -4708.001} C_VEL
LIN {X 0,Y 523.909,Z 285.221,A -85,B 0,C 180,E1 -4710.859,E2 -4710.859} C_VEL
LIN {X 0,Y 523.922,Z 285.223,A -85,B 0,C 180,E1 -4713.739,E2 -4713.739} C_VEL
LIN {X 0,Y 523.911,Z 285.219,A -85,B 0,C 180,E1 -4716.412,E2 -4716.412} C_VEL
LIN {X 0,Y 523.942,Z 285.217,A -85,B 0,C 180,E1 -4719.083,E2 -4719.083} C_VEL
LIN {X 0,Y 523.949,Z 285.219,A -85,B 0,C 180,E1 -4721.318,E2 -4721.318} C_VEL
LIN {X 0,Y 523.924,Z 285.219,A -85,B 0,C 180,E1 -4724.695,E2 -4724.695} C_VEL
LIN {X 0,Y 523.937,Z 285.225,A -85,B 0,C 180,E1 -4727.887,E2 -4727.887} C_VEL
LIN {X 0,Y 523.935,Z 285.217,A -85,B 0,C 180,E1 -4730.923,E2 -4730.923} C_VEL
LIN {X 0,Y 523.908,Z 285.227,A -85,B 0,C 180,E1 -4733.832,E2 -4733.832} C_VEL
LIN {X 0,Y 523.924,Z 285.221,A -85,B 0,C 180,E1 -4736.64,E2 -4736.64} C_VEL
LIN {X 0,Y 523.946,Z 285.22,A -85,B 0,C 180,E1 -4739.36,E2 -4739.36} C_VEL
LIN {X 0,Y 523.965,Z 285.22,A -85,B 0,C 180,E1 -4742.284,E2 -4742.284} C_VEL
LIN {X 0,Y 523.946,Z 285.222,A -85,B 0,C 180,E1 -4744.586,E2 -4744.586} C_VEL
LIN {X 0,Y 524.024,Z 285.414,A -85,B 0,C 180,E1 -4745.596,E2 -4745.596} C_VEL
LIN {X 0,Y 525.336,Z 293.853,A -85,B 0,C 180,E1 -4746.968,E2 -4746.968} C_VEL
LIN {X 0,Y 524.934,Z 313.86,A -85,B 0,C 180,E1 -4750.042,E2 -4750.042} C_VEL
LIN {X 0,Y 524.456,Z 333.709,A -85,B 0,C 180,E1 -4753.058,E2 -4753.058} C_VEL
LIN {X 0,Y 524.267,Z 345.526,A -85,B 0,C 180,E1 -4754.838,E2 -4754.838} C_VEL
LIN {X 0,Y 525.942,Z 357.971,A -85,B 0,C 180,E1 -4755.065,E2 -4755.065} C_VEL
LIN {X 0,Y 525.485,Z 453.706,A -85,B 0,C 180,E1 -4756.394,E2 -4756.394} C_VEL
LIN {X 0,Y 525.245,Z 467.096,A -85,B 0,C 180,E1 -4756.732,E2 -4756.732} C_VEL
LIN {X 0,Y 524.939,Z 480.456,A -85,B 0,C 180,E1 -4757.241,E2 -4757.241} C_VEL
LIN {X 0,Y 524.805,Z 492.013,A -85,B 0,C 180,E1 -4757.848,E2 -4757.848} C_VEL
LIN {X 0,Y 524.518,Z 503.316,A -85,B 0,C 180,E1 -4758.605,E2 -4758.605} C_VEL
LIN {X 0,Y 524.214,Z 513.798,A -85,B 0,C 180,E1 -4759.478,E2 -4759.478} C_VEL
LIN {X 0,Y 523.982,Z 522.37,A -85,B 0,C 180,E1 -4760.352,E2 -4760.352} C_VEL
LIN {X 0,Y 523.808,Z 530.279,A -85,B 0,C 180,E1 -4761.322,E2 -4761.322} C_VEL
LIN {X 0,Y 523.6,Z 538.001,A -85,B 0,C 180,E1 -4762.483,E2 -4762.483} C_VEL
LIN {X 0,Y 523.518,Z 543.16,A -85,B 0,C 180,E1 -4763.424,E2 -4763.424} C_VEL
LIN {X 0,Y 523.461,Z 548.422,A -85,B 0,C 180,E1 -4764.61,E2 -4764.61} C_VEL
LIN {X 0,Y 523.423,Z 552.403,A -85,B 0,C 180,E1 -4765.768,E2 -4765.768} C_VEL
LIN {X 0,Y 523.367,Z 555.341,A -85,B 0,C 180,E1 -4766.924,E2 -4766.924} C_VEL
LIN {X 0,Y 523.334,Z 556.739,A -85,B 0,C 180,E1 -4767.694,E2 -4767.694} C_VEL
LIN {X 0,Y 523.25,Z 558.344,A -85,B 0,C 180,E1 -4769.233,E2 -4769.233} C_VEL
LIN {X 0,Y 523.25,Z 558.561,A -85,B 0,C 180,E1 -4770.003,E2 -4770.003} C_VEL
LIN {X 0,Y 523.274,Z 557.737,A -85,B 0,C 180,E1 -4771.542,E2 -4771.542} C_VEL
LIN {X 0,Y 523.334,Z 556.741,A -85,B 0,C 180,E1 -4772.311,E2 -4772.311} C_VEL
LIN {X 0,Y 523.368,Z 555.343,A -85,B 0,C 180,E1 -4773.081,E2 -4773.081} C_VEL
LIN {X 0,Y 523.424,Z 552.402,A -85,B 0,C 180,E1 -4774.237,E2 -4774.237} C_VEL
LIN {X 0,Y 523.462,Z 548.419,A -85,B 0,C 180,E1 -4775.395,E2 -4775.395} C_VEL
LIN {X 0,Y 523.516,Z 542.31,A -85,B 0,C 180,E1 -4776.744,E2 -4776.744} C_VEL
LIN {X 0,Y 523.663,Z 535.594,A -85,B 0,C 180,E1 -4777.909,E2 -4777.909} C_VEL
LIN {X 0,Y 523.851,Z 527.287,A -85,B 0,C 180,E1 -4779.072,E2 -4779.072} C_VEL
LIN {X 0,Y 524.065,Z 518.767,A -85,B 0,C 180,E1 -4780.042,E2 -4780.042} C_VEL
LIN {X 0,Y 524.362,Z 508.242,A -85,B 0,C 180,E1 -4781.012,E2 -4781.012} C_VEL
LIN {X 0,Y 524.633,Z 497.921,A -85,B 0,C 180,E1 -4781.783,E2 -4781.783} C_VEL
LIN {X 0,Y 524.899,Z 486.405,A -85,B 0,C 180,E1 -4782.47,E2 -4782.47} C_VEL
LIN {X 0,Y 525.121,Z 474.644,A -85,B 0,C 180,E1 -4783.005,E2 -4783.005} C_VEL
LIN {X 0,Y 525.341,Z 461.088,A -85,B 0,C 180,E1 -4783.443,E2 -4783.443} C_VEL
LIN {X 0,Y 525.555,Z 447.491,A -85,B 0,C 180,E1 -4783.708,E2 -4783.708} C_VEL
LIN {X 0,Y 525.81,Z 355.583,A -85,B 0,C 180,E1 -4784.974,E2 -4784.974} C_VEL
LIN {X 0,Y 524.31,Z 345.614,A -85,B 0,C 180,E1 -4785.179,E2 -4785.179} C_VEL
LIN {X 0,Y 524.752,Z 323.724,A -85,B 0,C 180,E1 -4788.528,E2 -4788.528} C_VEL
LIN {X 0,Y 525.179,Z 305.22,A -85,B 0,C 180,E1 -4791.388,E2 -4791.388} C_VEL
LIN {X 0,Y 525.459,Z 293.472,A -85,B 0,C 180,E1 -4793.24,E2 -4793.24} C_VEL
LIN {X 0,Y 523.976,Z 285.217,A -85,B 0,C 180,E1 -4794.65,E2 -4794.65} C_VEL
